      sAdsIkInkStorageTank[iL_Counter].sI_EnableMaintenance.bO_CommandCanEx  :=     sAdsIkInkStorageTank[iL_Counter].sI_EnableBalance.bI_Command
                                                                                AND NOT sAdsIkInkStorageTank[iL_Counter].sI_EnableMaintenance.bI_Command
                                                                                AND NOT sAdsIkInkStorageTank[iL_Counter].sI_EnableMaintenance.bO_CommandExec;
(*      bL_MessageWarning[iL_Counter] := (   sAdsIkInkStorageTank[iL_Counter].bO_StorageTankWarning
                                        OR (    sAdsIkInkStorageTank[iL_Counter].bO_StorageTankError
                                            AND NOT sAdsIkInkStorageTank[iL_Counter].bI_EnableStorageTank));*)
      bL_MessageWarning[iL_Counter] := (    sAdsIkInkStorageTank[iL_Counter].bO_StorageTankWarning
                                        AND sAdsIkInkStorageTank[iL_Counter].bI_EnableStorageTank);
      bL_MessageError  [iL_Counter] := (    sAdsIkInkStorageTank[iL_Counter].bO_StorageTankError
                                        AND sAdsIkInkStorageTank[iL_Counter].bI_EnableStorageTank);
    END_FOR; (*FOR iL_Counter := 1 TO iCIk_NB_INKBALANCE DO*)

    FOR iL_Counter := 1 TO iCIk_NB_INKSTORAGE_TANK DO
      (*Storage Messages*)
      fB_BalanceMsgHandler[iL_Counter]();	(*Call to check for blocked access*)

      fb_BalanceMsg[iL_Counter, 1](bI_Status := fb_BalanceLink.wO_ErrorCodeChannel[iL_Counter].1);
      fb_BalanceMsg[iL_Counter, 2](bI_Status := fb_BalanceLink.wO_ErrorCodeChannel[iL_Counter].2);
      fb_BalanceMsg[iL_Counter, 3](bI_Status := fb_BalanceLink.wO_ErrorCodeChannel[iL_Counter].3);
      fb_BalanceMsg[iL_Counter, 4](bI_Status := fb_BalanceLink.wO_ErrorCodeChannel[iL_Counter].4);
      fb_BalanceMsg[iL_Counter, 5](bI_Status := FALSE);
      fb_BalanceMsg[iL_Counter, 6](bI_Status := FALSE);
      fb_BalanceMsg[iL_Counter, 7](bI_Status := FALSE);
      fb_BalanceMsg[iL_Counter, 8](bI_Status := bL_MessageWarning[iL_Counter]);
      fb_BalanceMsg[iL_Counter, 9](bI_Status := bL_MessageError  [iL_Counter]);
      fb_BalanceMsg[iL_Counter,10](bI_Status := FALSE);
      fb_BalanceMsg[iL_Counter,11](bI_Status := FALSE);  (*InkStorageTankMixerNotWorking*)
      (*Storage tank level info message*)
      fb_BalanceMsg[iL_Counter,12](bI_Status :=     (   sAdsIkInkStorageTank[iL_Counter].bO_StorageTankWarning
                                                     OR sAdsIkInkStorageTank[iL_Counter].bO_StorageTankError)
                                                AND NOT sAdsIkInkStorageTank[iL_Counter].cO_StatusStorageTank.eO_Activ);
      fB_BalanceMsg[iL_Counter,13](bI_Status :=     fb_BarcodeStoragetank.bO_LabelScanNeeded[iL_Counter]
                                                AND sAdsIkInkStorageTank[iL_Counter].cO_StatusStorageTank.eO_Activ);
      fB_BalanceMsg[iL_Counter,14](bI_Status :=     fb_BarcodeStoragetank.bO_LabelScanFalse [iL_Counter]
                                                AND sAdsIkInkStorageTank[iL_Counter].cO_StatusStorageTank.eO_Activ);
      fB_BalanceMsg[iL_Counter,15](bI_Status :=     NOT fb_Storagetank[iL_Counter].bI_HtAssignedToStorage
                                                AND sAdsIkInkStorageTank[iL_Counter].cO_StatusStorageTank.eO_Activ);

      fb_MsgQueueStorage[iL_Counter]();

    END_FOR;
  END_IF; (*IF bCIk_BALANCE_EXISTING THEN*)

  (*Set fO_StorageTankLevelPercent of conservation tank with bO_TankCleanerLevelEmpty*)
  IF bO_TankCleanerLevelEmpty THEN
    sAdsIkInkStorageTank[iCIk_NB_INKSTORAGE_TANK].fO_StorageTankLevelPercent.fO_Val := 0;
  ELSE
    sAdsIkInkStorageTank[iCIk_NB_INKSTORAGE_TANK].fO_StorageTankLevelPercent.fO_Val := 100;
END_IF
  
END_IF; (*Else when init Ok*)


(*Global status*)
bO_InkSystemOk :=     bO_VacuumOk
                  AND bO_TemperatureOk
                //AND bO_StorageTankOk
                  AND (NOT bO_CommandPrintlineExec[1] OR NOT bL_Engaged[1])
                  AND (NOT bO_CommandPrintlineExec[2] OR NOT bL_Engaged[2]);

IF sL_SystemCmd.bSleep THEN
  bO_InkStorageTankOk := TRUE;
ELSE
  bO_InkStorageTankOk := FALSE;
  FOR iL_Counter := 1 TO iCIk_NB_INKSTORAGE_TANK DO
    IF bCIk_INKSTORAGE_TANK_EXIST[iL_Counter] THEN
      bO_InkStorageTankOk := bO_InkStorageTankOk OR sAdsIkInkStorageTank[iL_Counter].bI_EnableStorageTank;
    END_IF;
  END_FOR;
END_IF;

(*WcState: 0 = Data valid, 1 = Data invalid*)
bO_TotalWcState     :=     bI_Pressure1WcState
                        OR bI_Pressure2WcState
                        OR bI_SubPressureWcState[1]
                        OR bI_Temperature1WcState
                        OR bI_InkLevel1WcState;


(********************************* END OF PRG ****************************************************)

ACTION AutoFlushingDevice:
IF aI_FlushingSafePattern = 'SAFE' THEN
  bL_FlushingUnlock      := TRUE;
ELSE
  aI_FlushingSafePattern := 'LOCKED';
  bL_FlushingUnlock      := FALSE;
END_IF;
fb_FTrigFlushingActive(CLK:= bL_FlushingActive);
fb_TonFlushingUnlock(IN := bL_FlushingUnlock AND (iL_FlushingState = 0), PT := T#180S);
IF fb_TonFlushingUnlock.Q OR fb_FTrigFlushingActive.Q THEN
  aI_FlushingSafePattern := 'LOCKED';
  bL_FlushingHtEmpty     := FALSE;
END_IF

fb_FlushingReturnFlowTimer( bI_Reset    := (iL_FlushingState = 0)
                          , bI_In       :=    fb_ReturnFlow[iCIk_MAP_HEADERTANK_RETURN_FLOW[PRG_INK.iL_SelHeaderTankFlushing]].fb_ReturnFlowPump.bOKp_EnablePump
                                           OR bO_FlushingReturnPump[iCIk_MAP_HEADERTANK_RETURN_FLOW[PRG_INK.iL_SelHeaderTankFlushing]]
                          , lIO_Seconds := lL_OpCounterReturnFlowSeconds
                          , lIO_Cycles  := lL_OpCounterReturnFlowCycles);

(*Return if function is not unlocked.*)
IF NOT bL_FlushingUnlock THEN
  RETURN;
END_IF

CASE iL_FlushingState OF
0:  (*Idle*)
  aL_FlushingState := 'Idle';

  IF     bL_FlushingActivate 
     AND bL_FlushingHtEmpty 
     AND sAdsIkHeaderTank[PRG_INK.iL_SelHeaderTankFlushing].sI_ActivateCleaner.bO_CommandCanEx
     AND NOT sAdsIkHeaderTank[PRG_INK.iL_SelHeaderTankFlushing].bI_EnableFillInk
  THEN
    bL_FlushingActive := TRUE;

    iL_FlushingState  := 1;
  ELSE
    bL_FlushingStop     := FALSE;
    bL_FlushingActivate := FALSE;
    bL_FlushingActive   := FALSE;
    bL_FlushingActiveHt         [PRG_INK.iL_SelHeaderTankFlushing] := FALSE;
    bL_FlushingReturnFlowRequest[PRG_INK.iL_SelHeaderTankFlushing] := FALSE;
    sAdsIkHeaderTank[PRG_INK.iL_SelHeaderTankFlushing].sI_ActivateCleaner.bI_Command := FALSE;
	END_IF

1:  (*Start fill cleaner*)
  aL_FlushingState := 'Start fill cleaner';

  sAdsIkHeaderTank[PRG_INK.iL_SelHeaderTankFlushing].sI_ActivateCleaner.bI_Command := TRUE;
  
  IF sAdsIkHeaderTank[PRG_INK.iL_SelHeaderTankFlushing].sI_ActivateCleaner.bO_CommandExec THEN
    sAdsIkHeaderTank[PRG_INK.iL_SelHeaderTankFlushing].sI_ActivateCleaner.bI_Command := FALSE;
    bL_FlushingActiveHt[PRG_INK.iL_SelHeaderTankFlushing] := TRUE;

    iL_FlushingState := 2;
	END_IF
  
  IF bL_FlushingStop THEN
    sAdsIkHeaderTank[PRG_INK.iL_SelHeaderTankFlushing].sI_ActivateCleaner.bI_Command := FALSE;

    iL_FlushingState := 5;
	END_IF
  
2:  (*Fill cleaner*)
  aL_FlushingState := 'Fill cleaner';

  IF NOT sAdsIkHeaderTank[PRG_INK.iL_SelHeaderTankFlushing].sI_ActivateCleaner.bO_CommandExec THEN
    iL_FlushingState := 3;
	END_IF
  
  IF bL_FlushingStop THEN
    iL_FlushingState := 5;
	END_IF
  
3:  (*Start empty cleaner*)
  aL_FlushingState := 'Start empty cleaner';

  bL_FlushingReturnFlowRequest[PRG_INK.iL_SelHeaderTankFlushing] := TRUE;
  
  IF    fb_ReturnFlow[iCIk_MAP_HEADERTANK_RETURN_FLOW[PRG_INK.iL_SelHeaderTankFlushing]].fb_ReturnFlowPump.bOKp_EnablePump 
     OR bO_FlushingReturnPump[iCIk_MAP_HEADERTANK_RETURN_FLOW[PRG_INK.iL_SelHeaderTankFlushing]]
  THEN
    iL_FlushingState := 4;
	END_IF

  IF bL_FlushingStop THEN
    bL_FlushingReturnFlowRequest[PRG_INK.iL_SelHeaderTankFlushing] := FALSE;

    iL_FlushingState := 5;
	END_IF
  
4:  (*Empty cleaner*)
  aL_FlushingState := 'Empty cleaner';

  IF lL_OpCounterReturnFlowSeconds >= lL_TimeFlushingReturnFlow THEN
    bL_FlushingReturnFlowRequest[PRG_INK.iL_SelHeaderTankFlushing] := FALSE;
    bL_FlushingActiveHt         [PRG_INK.iL_SelHeaderTankFlushing] := FALSE;

    iL_FlushingState := 0;
	END_IF

  IF bL_FlushingStop THEN
    bL_FlushingReturnFlowRequest[PRG_INK.iL_SelHeaderTankFlushing] := FALSE;

    iL_FlushingState := 5;
	END_IF
  
5:  (*Abort*)
  aL_FlushingState := 'Abort';

  IF     NOT sAdsIkHeaderTank[PRG_INK.iL_SelHeaderTankFlushing].sI_ActivateCleaner.bO_CommandExec
     AND (   NOT fb_ReturnFlow[iCIk_MAP_HEADERTANK_RETURN_FLOW[PRG_INK.iL_SelHeaderTankFlushing]].fb_ReturnFlowPump.bOKp_EnablePump
          OR NOT bO_FlushingReturnPump[iCIk_MAP_HEADERTANK_RETURN_FLOW[PRG_INK.iL_SelHeaderTankFlushing]])
  THEN
    bL_FlushingStop     := FALSE;
    bL_FlushingActivate := FALSE;

    iL_FlushingState := 0;
	END_IF

END_CASE
END_ACTION

ACTION Init:
(*************************************************************************************************)
(* --- Module preprarations --- *)


(*GENERAL*)
(*************************************************************************************************)
(*System init*)
CASE cL_State OF

  cL_INIT : 		(*First init*)

                // Get system reference
                ISystemBase := PRG_SYSTEMBASE.getSystemBaseInterface();
                IF ISystemBase = 0 THEN RETURN; END_IF
                // Wait until system(base) is booted
                IF ISystemBase.bBooting THEN RETURN; END_IF
                
                // Command / Status interface
                PRG_SYSTEMBASE.getSystemCmdStatusInterface(iSystemCmd=>iSystemCmd, iSystemStatus=>iSystemStatus);
                
                // Build mapping information for ADS
                Mapping();
                
                // Register module to system
                pModuleDef := ISystemBase.regModule(
                  pAdsInfo:=ADR(sC_Ads_Info),
                  pMapInfo:=ADR(sMappingInfo)
                );
                IF pModuleDef = 0 THEN RETURN; END_IF

                Fb_RegToAry.iI_ActElem := 0;   (*init module's block mapping array*)
                Fb_RegToAry.sI_Parent := FC_CREATE_ARYPTR(ADR(sL_MOD_MAP), SIZEOF(sL_MOD_MAP)/SIZEOF(sL_MOD_MAP[1]), SIZEOF(sL_MOD_MAP[1]));

                iMachineInk[1] := PRG_MACHINE.fb_InterfaceMachineInk[1];
                iMachineInk[2] := PRG_MACHINE.fb_InterfaceMachineInk[2];

                cL_State := cL_INIT_PRG;

  cL_INIT_PRG :	(*Program call init*)

                FOR iL_CounterDgas := 1 TO iCIk_NB_DGAS DO
                  ;
                END_FOR;

                FOR iL_CounterMenc := 1 TO iCIk_NB_MENC DO
                  ;
                END_FOR

                FOR iL_CounterSubMenc := 1 TO iCIk_NB_SUB_MENC DO
                  ;
                END_FOR

                bL_RemVar_Init := TRUE;    (* Write variables by remanent variables *)
                RemVar();

                cL_State := cL_INIT_OK;

  cL_INIT_OK: 	(*First init ok*)
                bO_InitOk := TRUE;

END_CASE;



(*************************************************************************************************)
(*ADS Structures Init*)
(*************************************************************************************************)

(*INK TABLE*)
(*************************************************************************************************)
sL_InkTable[1].iI_ColorID := 0; sL_InkTable[1].aI_ColorName := sC_Config_I.aC_HEADERTANK_NAME_DETAIL[1]; sL_InkTable[1].lI_ColorRGB := 16#FFFFFF;
sL_InkTable[2].iI_ColorID := 0; sL_InkTable[2].aI_ColorName := sC_Config_I.aC_HEADERTANK_NAME_DETAIL[2]; sL_InkTable[2].lI_ColorRGB := 16#FFFFFF;
sL_InkTable[3].iI_ColorID := 1; sL_InkTable[3].aI_ColorName := sC_Config_I.aC_HEADERTANK_NAME_DETAIL[3]; sL_InkTable[3].lI_ColorRGB := 16#FFFFFF;
sL_InkTable[4].iI_ColorID := 1; sL_InkTable[4].aI_ColorName := sC_Config_I.aC_HEADERTANK_NAME_DETAIL[4]; sL_InkTable[4].lI_ColorRGB := 16#FFFFFF;


(*DEGASSING*)
(*************************************************************************************************)
(*Pneumatic Controller Board CB1*)
(*generate block ads name*)
FOR iL_Counter := 1 TO iCIk_NB_DGAS DO
  aL_Name := sC_Config_I.aC_DGAS_NAME;
  IF sC_Config_I.aC_DGAS_NAME_DETAIL[iL_Counter] <> '' THEN
    aL_Name := CONCAT(aL_Name, CONCAT(' - ', sC_Config_I.aC_DGAS_NAME_DETAIL[iL_Counter]));
  ELSE
    aL_Name := CONCAT(aL_Name, INT_TO_STRING(iL_Counter));
  END_IF
  sAdsIkDgas[iL_Counter].aO_Name := aL_Name;
END_FOR;

sAdsIkDgas[eIk_DGAS1].sI_PressSet.aC_Type := sC_Config_I.aC_DGAS1_PRESS_TYPE;
sAdsIkDgas[eIk_DGAS1].sI_PressSet.aC_Unit := sC_Config_I.aC_DGAS1_PRESS_UNIT;
sAdsIkDgas[eIk_DGAS1].sI_PressSet.fC_Min  := sC_Config_I.fL_DGAS1_PRESS_SET_MIN;
sAdsIkDgas[eIk_DGAS1].sI_PressSet.fC_Max  := sC_Config_I.fL_DGAS1_PRESS_SET_MAX;

sAdsIkDgas[eIk_DGAS1].sO_PressAct.aC_Type := sC_Config_I.aC_DGAS1_PRESS_TYPE;
sAdsIkDgas[eIk_DGAS1].sO_PressAct.aC_Unit := sC_Config_I.aC_DGAS1_PRESS_UNIT;
sAdsIkDgas[eIk_DGAS1].sO_PressAct.fC_Min  := sC_Config_I.fL_DGAS1_PRESS_ACT_MIN;
sAdsIkDgas[eIk_DGAS1].sO_PressAct.fC_Max  := sC_Config_I.fL_DGAS1_PRESS_ACT_MAX;

sAdsIkDgas[eIk_DGAS1].sI_AckPression.bO_CommandExist := TRUE;


(*MENISCUS*)
(*************************************************************************************************)
(*generate block ads name*)
FOR iL_Counter := 1 TO iCIk_NB_MENC DO
  aL_Name := sC_Config_I.aC_MENC_NAME;
  IF sC_Config_I.aC_MENC_NAME_DETAIL[iL_Counter] <> '' THEN
    aL_Name := CONCAT(aL_Name, CONCAT(' - ', sC_Config_I.aC_MENC_NAME_DETAIL[iL_Counter]));
  ELSE
    aL_Name := CONCAT(aL_Name, INT_TO_STRING(iL_Counter));
  END_IF
  sAdsIkMenc[iL_Counter].aO_Name := aL_Name;

  sAdsIkMenc[iL_Counter].sI_PressSet.aC_Type := sC_Config_I.aC_MENC_PRESS_TYPE;
  sAdsIkMenc[iL_Counter].sI_PressSet.aC_Unit := sC_Config_I.aC_MENC_PRESS_UNIT;
  sAdsIkMenc[iL_Counter].sI_PressSet.fC_Min  := sC_Config_I.fL_MENC_PRESS_SET_MIN;
  sAdsIkMenc[iL_Counter].sI_PressSet.fC_Max  := sC_Config_I.fL_MENC_PRESS_SET_MAX;

  sAdsIkMenc[iL_Counter].sO_PressAct.aC_Type := sC_Config_I.aC_MENC_PRESS_TYPE;
  sAdsIkMenc[iL_Counter].sO_PressAct.aC_Unit := sC_Config_I.aC_MENC_PRESS_UNIT;
  sAdsIkMenc[iL_Counter].sO_PressAct.fC_Min  := sC_Config_I.fL_MENC_PRESS_ACT_MIN;
  sAdsIkMenc[iL_Counter].sO_PressAct.fC_Max  := sC_Config_I.fL_MENC_PRESS_ACT_MAX;

  sAdsIkMenc[iL_Counter].sI_AckPression.bO_CommandExist := TRUE;
END_FOR;


(*SUB MENISCUS*)
(*************************************************************************************************)
(*Sub meniscus starts behind the meniscus*)
(*generate block ads name*)
FOR iL_CounterSubMenc := 1 TO iCIk_NB_SUB_MENC DO
  aL_Name := sC_Config_I.aC_SUB_MENC_NAME;
  IF sC_Config_I.aC_SUB_MENC_NAME_DETAIL[iL_CounterSubMenc] <> '' THEN
    aL_Name := CONCAT(aL_Name, CONCAT(' - ', sC_Config_I.aC_SUB_MENC_NAME_DETAIL[iL_CounterSubMenc]));
  ELSE
    aL_Name := CONCAT(aL_Name, INT_TO_STRING(iCIk_NB_MENC + iL_CounterSubMenc));
  END_IF
  sAdsIkMenc[iCIk_NB_MENC + iL_CounterSubMenc].aO_Name := aL_Name;

  sAdsIkMenc[iCIk_NB_MENC + iL_CounterSubMenc].sI_PressSet.aC_Type := sC_Config_I.aC_SUB_MENC_PRESS_TYPE;
  sAdsIkMenc[iCIk_NB_MENC + iL_CounterSubMenc].sI_PressSet.aC_Unit := sC_Config_I.aC_SUB_MENC_PRESS_UNIT;
  sAdsIkMenc[iCIk_NB_MENC + iL_CounterSubMenc].sI_PressSet.fC_Min  := sC_Config_I.fL_SUB_MENC_PRESS_SET_MIN;
  sAdsIkMenc[iCIk_NB_MENC + iL_CounterSubMenc].sI_PressSet.fC_Max  := sC_Config_I.fL_SUB_MENC_PRESS_SET_MAX;

  sAdsIkMenc[iCIk_NB_MENC + iL_CounterSubMenc].sO_PressAct.aC_Type := sC_Config_I.aC_SUB_MENC_PRESS_TYPE;
  sAdsIkMenc[iCIk_NB_MENC + iL_CounterSubMenc].sO_PressAct.aC_Unit := sC_Config_I.aC_SUB_MENC_PRESS_UNIT;
  sAdsIkMenc[iCIk_NB_MENC + iL_CounterSubMenc].sO_PressAct.fC_Min  := sC_Config_I.fL_SUB_MENC_PRESS_ACT_MIN;
  sAdsIkMenc[iCIk_NB_MENC + iL_CounterSubMenc].sO_PressAct.fC_Max  := sC_Config_I.fL_SUB_MENC_PRESS_ACT_MAX;

  sAdsIkMenc[iCIk_NB_MENC + iL_CounterSubMenc].sI_AckPression.bO_CommandExist := TRUE;

  //sAdsIkMenc[iCIk_NB_MENC + iL_CounterSubMenc].iO_ColorId          := x;
END_FOR;


(*PURGE*)
(*************************************************************************************************)
(*generate block ads name*)
FOR iL_Counter := 1 TO iCIk_NB_PURGE_CONTR DO
  aL_Name := sC_Config_I.aC_PURGE_NAME;
  IF sC_Config_I.aC_PURGE_NAME_DETAIL[iL_Counter] <> '' THEN
    aL_Name := CONCAT(aL_Name, CONCAT(' - ', sC_Config_I.aC_PURGE_NAME_DETAIL[iL_Counter]));
  ELSE
    aL_Name := CONCAT(aL_Name, INT_TO_STRING(iL_Counter));
  END_IF
  sAdsIkPurgeController[iL_Counter].aO_Name := aL_Name;

  sAdsIkPurgeController[iL_Counter].sI_ActivatePurge.bO_CommandCanEx := TRUE;
  sAdsIkPurgeController[iL_Counter].sI_ActivatePurge.bO_CommandExist := TRUE;
END_FOR;

FOR iL_Counter := 1 TO iCIk_NB_PURGE_GROUP DO
  (*generate block ads name*)
  aL_Name := sC_Config_I.aC_PURGE_GROUP_NAME;
  IF sC_Config_I.aC_PURGE_GROUP_NAME_DETAIL[iL_Counter] <> '' THEN
    aL_Name := CONCAT(aL_Name, CONCAT(' - ', sC_Config_I.aC_PURGE_GROUP_NAME_DETAIL[iL_Counter]));
  ELSE
    aL_Name := CONCAT(aL_Name, INT_TO_STRING(iL_Counter));
  END_IF
  sAdsIkPurgeGroup[iL_Counter].aO_Name := aL_Name;

  sAdsIkPurgeGroup[iL_Counter].cO_Status.eO_Avbl      := TRUE;
  sAdsIkPurgeGroup[iL_Counter].cO_ValveStatus.eO_Avbl := TRUE;
END_FOR


(*INK*)
(*************************************************************************************************)
FOR iL_Counter := 1 TO iCIk_NB_INK_PUMPS DO
  (*generate block ads name*)
  aL_Name := sC_Config_I.aC_INKPUMP_NAME;
  IF sC_Config_I.aC_INKPUMP_NAME_DETAIL[iL_Counter] <> '' THEN
    aL_Name := CONCAT(aL_Name, CONCAT(' - ', sC_Config_I.aC_INKPUMP_NAME_DETAIL[iL_Counter]));
  ELSE
    aL_Name := CONCAT(aL_Name, INT_TO_STRING(iL_Counter));
  END_IF
  sAdsIkInkPump[iL_Counter].aO_Name := aL_Name;

  sAdsIkInkPump[iL_Counter].sI_InkPumpSpeedSet.aC_Type := sC_Config_I.aC_INKPUMP_SPEED_TYPE;
  sAdsIkInkPump[iL_Counter].sI_InkPumpSpeedSet.aC_Unit := sC_Config_I.aC_INKPUMP_SPEED_UNIT;
  sAdsIkInkPump[iL_Counter].sI_InkPumpSpeedSet.lC_Min  := sC_Config_I.lL_INKPUMP_SPEED_SET_MIN;
  sAdsIkInkPump[iL_Counter].sI_InkPumpSpeedSet.lC_Max  := sC_Config_I.lL_INKPUMP_SPEED_SET_MAX;
END_FOR

FOR iL_Counter := 1 TO iCIk_NB_HEADERTANK DO
  (*IF bCIk_HEADERTANK_EXIST[iL_Counter] THEN*)
    (*generate block ads name*)
    aL_Name := sC_Config_I.aC_HEADERTANK_NAME;
    IF sC_Config_I.aC_HEADERTANK_NAME_DETAIL[iL_Counter] <> '' THEN
      aL_Name := CONCAT(aL_Name, CONCAT(' - ', sC_Config_I.aC_HEADERTANK_NAME_DETAIL[iL_Counter]));
    ELSE
      aL_Name := CONCAT(aL_Name, INT_TO_STRING(iL_Counter));
    END_IF
    sAdsIkHeaderTank[iL_Counter].aO_Name := aL_Name;

		sAdsIkHeaderTank[iL_Counter].sI_StoragetankAssignment.bC_Exist    := TRUE;
		sAdsIkHeaderTank[iL_Counter].sO_ActStoragetankAssignment.bC_Exist := TRUE;

		(*un-/fill ink*)
		sAdsIkHeaderTank[iL_Counter].bO_EnableFillInkCanEn               := bCIk_HEADERTANK_EXIST[iL_Counter];
		sAdsIkHeaderTank[iL_Counter].bO_EnableUnFillInkCanEn             := bCIk_HEADERTANK_EXIST[iL_Counter];
		sAdsIkHeaderTank[iL_Counter].cO_StatusFillInk.eO_Avbl            := bCIk_HEADERTANK_EXIST[iL_Counter];
		sAdsIkHeaderTank[iL_Counter].cO_StatusUnFillInk.eO_Avbl          := bCIk_HEADERTANK_EXIST[iL_Counter];

		sAdsIkHeaderTank[iL_Counter].sI_ActivateCleaner.bO_CommandCanEx  := bCIk_HEADERTANK_FILL_CLEANER[iL_Counter];
		sAdsIkHeaderTank[iL_Counter].sI_ActivateRefuse.bO_CommandCanEx   := bCIk_HEADERTANK_REFUSE      [iL_Counter];
		sAdsIkHeaderTank[iL_Counter].sI_ActivateExchange.bO_CommandCanEx := FALSE;

		sAdsIkHeaderTank[iL_Counter].sI_ActivateCleaner.bO_CommandExist	 := bCIk_HEADERTANK_FILL_CLEANER[iL_Counter];
		sAdsIkHeaderTank[iL_Counter].sI_ActivateRefuse.bO_CommandExist	 := bCIk_HEADERTANK_REFUSE      [iL_Counter];
		sAdsIkHeaderTank[iL_Counter].sI_ActivateExchange.bO_CommandExist := FALSE;

    sAdsIkHeaderTank[iL_Counter].sI_CommandChange.bO_CommandExist    := bCIk_HEADERTANK_CHANGE      [iL_Counter];

		(*error ack exist*)
		sAdsIkHeaderTank[iL_Counter].sI_AckFillInk.bO_CommandExist       := TRUE;

		(*tank heater*)
		sAdsIkHeaderTank[iL_Counter].sI_TankHeaterSet.bC_Exist   := FALSE;
		sAdsIkHeaderTank[iL_Counter].sI_TankHeaterSet.aC_Type    := sC_Config_I.aC_TEMP_TYPE;
		sAdsIkHeaderTank[iL_Counter].sI_TankHeaterSet.aC_Unit    := sC_Config_I.aC_TEMP_UNIT;
		sAdsIkHeaderTank[iL_Counter].sI_TankHeaterSet.fC_Min     := sC_Config_I.fL_TEMP_SET_VAL_MIN;
		sAdsIkHeaderTank[iL_Counter].sI_TankHeaterSet.fC_Max     := sC_Config_I.fL_TEMP_SET_VAL_MAX;

		sAdsIkHeaderTank[iL_Counter].sO_TankHeaterAct.bC_Exist   := FALSE;
		sAdsIkHeaderTank[iL_Counter].sO_TankHeaterAct.aC_Type    := sC_Config_I.aC_TEMP_TYPE;
		sAdsIkHeaderTank[iL_Counter].sO_TankHeaterAct.aC_Unit    := sC_Config_I.aC_TEMP_UNIT;
    sAdsIkHeaderTank[iL_Counter].sO_TankHeaterAct.fC_Min     := sC_Config_I.fL_TEMP_ACT_VAL_MIN;
    sAdsIkHeaderTank[iL_Counter].sO_TankHeaterAct.fC_Max     := sC_Config_I.fL_TEMP_ACT_VAL_MAX;

		sAdsIkHeaderTank[iL_Counter].bO_EnableTankHeaterCanEn    := FALSE;
		sAdsIkHeaderTank[iL_Counter].cO_StatusTankHeater.eO_Avbl := FALSE;
	(*END_IF*)
END_FOR

FOR iL_Counter := 1 TO iCIk_NB_HEADERTANK_GROUP DO
  (*generate block ads name*)
  aL_Name := sC_Config_I.aC_HEADERTANKGROUP_NAME;
  IF sC_Config_I.aC_HEADERTANKGROUP_NAME_DETAIL[iL_Counter] <> '' THEN
    aL_Name := CONCAT(aL_Name, CONCAT(' - ', sC_Config_I.aC_HEADERTANKGROUP_NAME_DETAIL[iL_Counter]));
  ELSE
    aL_Name := CONCAT(aL_Name, INT_TO_STRING(iL_Counter));
  END_IF
  sAdsIkHeaderTankGroup[iL_Counter].aO_Name := aL_Name;

  sAdsIkHeaderTankGroup[iL_Counter].sI_CommandChangeInk.bO_CommandExist := TRUE;
  sAdsIkHeaderTankGroup[iL_Counter].sI_CommandChangeInk.bO_CommandCanEx := TRUE;
  sAdsIkHeaderTankGroup[iL_Counter].sI_CommandEmptyInk.bO_CommandExist  := FALSE;
  sAdsIkHeaderTankGroup[iL_Counter].sI_CommandEmptyInk.bO_CommandCanEx  := FALSE;
END_FOR


(*TEMP*)
(*************************************************************************************************)
FOR iL_Counter := 1 TO iCIk_NB_TEMP_CONTR DO
  (*generate block ads name*)
  aL_Name := sC_Config_I.aC_TEMP_NAME;
  IF sC_Config_I.aC_TEMP_NAME_DETAIL[iL_Counter] <> '' THEN
    aL_Name := CONCAT(aL_Name, CONCAT(' - ', sC_Config_I.aC_TEMP_NAME_DETAIL[iL_Counter]));
  ELSE
    aL_Name := CONCAT(aL_Name, INT_TO_STRING(iL_Counter));
  END_IF
  sAdsIkHeater[iL_Counter].aO_Name := aL_Name;

  sAdsIkHeater[iL_Counter].sI_HeaterSet.aC_Type    := sC_Config_I.aC_TEMP_TYPE;
  sAdsIkHeater[iL_Counter].sI_HeaterSet.aC_Unit    := sC_Config_I.aC_TEMP_UNIT;
  sAdsIkHeater[iL_Counter].sI_HeaterSet.fC_Min     := sC_Config_I.fL_TEMP_SET_VAL_MIN;
  sAdsIkHeater[iL_Counter].sI_HeaterSet.fC_Max     := sC_Config_I.fL_TEMP_SET_VAL_MAX;

  sAdsIkHeater[iL_Counter].sO_HeaterAct.aC_Type    := sC_Config_I.aC_TEMP_TYPE;
  sAdsIkHeater[iL_Counter].sO_HeaterAct.aC_Unit    := sC_Config_I.aC_TEMP_UNIT;
  sAdsIkHeater[iL_Counter].sO_HeaterAct.fC_Min     := sC_Config_I.fL_TEMP_ACT_VAL_MIN;
  sAdsIkHeater[iL_Counter].sO_HeaterAct.fC_Max     := sC_Config_I.fL_TEMP_ACT_VAL_MAX;

  sAdsIkHeater[iL_Counter].bO_EnableHeaterCanEn    := TRUE;
  sAdsIkHeater[iL_Counter].cO_StatusHeater.eO_Avbl := TRUE;
END_FOR


(* STORAGE TANK *)
(**********************************************************************************)
FOR iL_Counter := 1 TO iCIk_NB_INKSTORAGE_TANK DO
  (*generate block ads name*)
  aL_Name := sC_Config_I.aC_STORAGETANK_NAME;
  IF sC_Config_I.aC_STORAGETANK_NAME_DETAIL[iL_Counter] <> '' THEN
    aL_Name := CONCAT(aL_Name, CONCAT(' - ', sC_Config_I.aC_STORAGETANK_NAME_DETAIL[iL_Counter]));
  ELSE
    aL_Name := CONCAT(aL_Name, INT_TO_STRING(iL_Counter));
  END_IF
  sAdsIkInkStorageTank[iL_Counter].aO_Name := aL_Name;

  (*Special storage tank for conservation*)
  IF sC_Config_I.aC_STORAGETANK_NAME_DETAIL[iL_Counter] = sC_Config_I.aC_STORAGETANK_CONSERVATION THEN
    sAdsIkInkStorageTank[iL_Counter].bO_EnableStorageTankCanEn             := FALSE;
    sAdsIkInkStorageTank[iL_Counter].cO_StatusStorageTank.eO_Avbl          := FALSE;
    sAdsIkInkStorageTank[iL_Counter].sI_EnableMaintenance.bO_CommandCanEx  := FALSE;
    sAdsIkInkStorageTank[iL_Counter].sI_EnableMaintenance.bO_CommandExist  := FALSE;
    sAdsIkInkStorageTank[iL_Counter].fO_StorageTankLevelLiter.bC_Exist     := FALSE;
    sAdsIkInkStorageTank[iL_Counter].sI_MaintenanceTimeout.bC_Exist        := FALSE;
    
    (*Varnish parameter*)
    sAdsIkInkStorageTank[iL_Counter].bO_InkParameterExist                  := FALSE;
    sAdsIkInkStorageTank[iL_Counter].sI_InkParameter.sTemperature.aC_Type  := sC_Config_I.aC_TEMP_TYPE;
    sAdsIkInkStorageTank[iL_Counter].sI_InkParameter.sTemperature.aC_Unit  := sC_Config_I.aC_TEMP_UNIT;
    sAdsIkInkStorageTank[iL_Counter].sI_InkParameter.sTemperature.fC_Min   := sC_Config_I.fL_TEMP_SET_VAL_MIN;
    sAdsIkInkStorageTank[iL_Counter].sI_InkParameter.sTemperature.fC_Max   := sC_Config_I.fL_TEMP_SET_VAL_MAX;
    sAdsIkInkStorageTank[iL_Counter].sI_InkParameter.sMeniscus.aC_Type     := sC_Config_I.aC_SUB_MENC_PRESS_TYPE;
    sAdsIkInkStorageTank[iL_Counter].sI_InkParameter.sMeniscus.aC_Unit     := sC_Config_I.aC_SUB_MENC_PRESS_UNIT;
    sAdsIkInkStorageTank[iL_Counter].sI_InkParameter.sMeniscus.fC_Min      := sC_Config_I.fL_SUB_MENC_PRESS_SET_MIN;
    sAdsIkInkStorageTank[iL_Counter].sI_InkParameter.sMeniscus.fC_Max      := sC_Config_I.fL_SUB_MENC_PRESS_SET_MAX;
    sAdsIkInkStorageTank[iL_Counter].sI_InkParameter.sDensity.aC_Unit      := sC_Config_I.aC_STORAGETANK_DENSITY;
    sAdsIkInkStorageTank[iL_Counter].sI_InkParameter.sViscosity.aC_Unit    := sC_Config_I.aC_STORAGETANK_VISCOSITY;

    sAdsIkInkStorageTank[iL_Counter].sI_EnableBalance.bO_CommandCanEx      := FALSE;
    sAdsIkInkStorageTank[iL_Counter].sI_EnableBalance.bO_CommandExist      := FALSE;
    sAdsIkInkStorageTank[iL_Counter].cO_StatusBalance.eO_Avbl              := FALSE;
    sAdsIkInkStorageTank[iL_Counter].bO_SetZeroCanEx                       := FALSE;
  ELSE
    sAdsIkInkStorageTank[iL_Counter].bI_EnableStorageTank                  := TRUE;
    sAdsIkInkStorageTank[iL_Counter].bO_EnableStorageTankCanEn             := TRUE;
    sAdsIkInkStorageTank[iL_Counter].cO_StatusStorageTank.eO_Avbl          := FALSE;
  
    sAdsIkInkStorageTank[iL_Counter].sI_EnableMaintenance.bO_CommandCanEx  := TRUE;
    sAdsIkInkStorageTank[iL_Counter].sI_EnableMaintenance.bO_CommandExist  := TRUE;
  
    sAdsIkInkStorageTank[iL_Counter].fO_StorageTankLevelLiter.aC_Type      := sC_Config_I.aC_STORAGETANK_TYPE;
    sAdsIkInkStorageTank[iL_Counter].fO_StorageTankLevelLiter.aC_Unit      := sC_Config_I.aC_STORAGETANK_UNITLITER;
    sAdsIkInkStorageTank[iL_Counter].fO_StorageTankLevelPercent.aC_Type    := sC_Config_I.aC_STORAGETANK_TYPE;
    sAdsIkInkStorageTank[iL_Counter].fO_StorageTankLevelPercent.aC_Unit    := sC_Config_I.aC_STORAGETANK_UNITPERCENT;
  
    sAdsIkInkStorageTank[iL_Counter].sI_MaintenanceTimeout.aC_Type         := sC_Config_I.aC_STORAGETANK_MAINTENANCE_TYPE;
    sAdsIkInkStorageTank[iL_Counter].sI_MaintenanceTimeout.aC_Unit         := sC_Config_I.aC_STORAGETANK_MAINTENANCE_UNIT;
    sAdsIkInkStorageTank[iL_Counter].sI_MaintenanceTimeout.lC_Min          := sC_Config_I.lL_STORAGETANK_MAINTENANCE_SET_MIN;
    sAdsIkInkStorageTank[iL_Counter].sI_MaintenanceTimeout.lC_Max          := sC_Config_I.lL_STORAGETANK_MAINTENANCE_SET_MAX;
  
    (*Varnish parameter*)
    sAdsIkInkStorageTank[iL_Counter].bO_InkParameterExist                  := TRUE;
    sAdsIkInkStorageTank[iL_Counter].sI_InkParameter.sTemperature.aC_Type  := sC_Config_I.aC_TEMP_TYPE;
    sAdsIkInkStorageTank[iL_Counter].sI_InkParameter.sTemperature.aC_Unit  := sC_Config_I.aC_TEMP_UNIT;
    sAdsIkInkStorageTank[iL_Counter].sI_InkParameter.sTemperature.fC_Min   := sC_Config_I.fL_TEMP_SET_VAL_MIN;
    sAdsIkInkStorageTank[iL_Counter].sI_InkParameter.sTemperature.fC_Max   := sC_Config_I.fL_TEMP_SET_VAL_MAX;
    sAdsIkInkStorageTank[iL_Counter].sI_InkParameter.sMeniscus.aC_Type     := sC_Config_I.aC_SUB_MENC_PRESS_TYPE;
    sAdsIkInkStorageTank[iL_Counter].sI_InkParameter.sMeniscus.aC_Unit     := sC_Config_I.aC_SUB_MENC_PRESS_UNIT;
    sAdsIkInkStorageTank[iL_Counter].sI_InkParameter.sMeniscus.fC_Min      := sC_Config_I.fL_SUB_MENC_PRESS_SET_MIN;
    sAdsIkInkStorageTank[iL_Counter].sI_InkParameter.sMeniscus.fC_Max      := sC_Config_I.fL_SUB_MENC_PRESS_SET_MAX;
    sAdsIkInkStorageTank[iL_Counter].sI_InkParameter.sDensity.aC_Unit      := sC_Config_I.aC_STORAGETANK_DENSITY;
    sAdsIkInkStorageTank[iL_Counter].sI_InkParameter.sViscosity.aC_Unit    := sC_Config_I.aC_STORAGETANK_VISCOSITY;
  END_IF
END_FOR;

FOR iL_Counter := 1 TO iCIk_NB_INKSTORAGE_TANK DO
  (*Varnish parameter*)
  IF sAdsIkInkStorageTank[iL_Counter].bO_InkParameterExist THEN
    sAdsIkInkStorageTank[iL_Counter].sI_InkParameter.iScannerId          := sR_RemVar_I.lR_VarParamScannerId[iL_Counter];
    sAdsIkInkStorageTank[iL_Counter].sI_InkParameter.iIndex              := sR_RemVar_I.iR_VarParamIndex    [iL_Counter];
    sAdsIkInkStorageTank[iL_Counter].sI_InkParameter.sTemperature.fI_Val := sR_RemVar_I.fR_VarParamTemp     [iL_Counter];
    sAdsIkInkStorageTank[iL_Counter].sI_InkParameter.sMeniscus.fI_Val    := sR_RemVar_I.fR_VarParamMenc     [iL_Counter];
    sAdsIkInkStorageTank[iL_Counter].sI_InkParameter.aWaveform           := sR_RemVar_I.aR_VarParamWaveform [iL_Counter];
    sAdsIkInkStorageTank[iL_Counter].sI_InkParameter.iTimer              := sR_RemVar_I.iR_VarParamTimer    [iL_Counter];
    sAdsIkInkStorageTank[iL_Counter].sI_InkParameter.sDensity.fI_Val     := sR_RemVar_I.fR_VarParamDensity  [iL_Counter];
    sAdsIkInkStorageTank[iL_Counter].sI_InkParameter.sViscosity.fI_Val   := sR_RemVar_I.fR_VarParamViscosity[iL_Counter];
    sAdsIkInkStorageTank[iL_Counter].sI_InkParameter.iColorId            := sR_RemVar_I.iR_VarParamColorId  [iL_Counter];
    FOR iL_Counter2 := 1 TO 10 DO
      sAdsIkInkStorageTank[iL_Counter].sI_InkParameter.bCompatibility[iL_Counter2] := sR_RemVar_I.bR_VarParamCompatibility[iL_Counter, iL_Counter2];
    END_FOR;
  END_IF
END_FOR;


(* BALANCE *)
(*************************************************************************************************)
(* -------------- init of the channels -------------------- *)
FOR iL_Counter := 1 TO iCIk_NB_INKBALANCE DO
  sAdsIkInkStorageTank[iL_Counter].sI_EnableBalance.bI_Command      := TRUE;
	sAdsIkInkStorageTank[iL_Counter].sI_EnableBalance.bO_CommandCanEx := TRUE;
	sAdsIkInkStorageTank[iL_Counter].sI_EnableBalance.bO_CommandExist := TRUE;
	sAdsIkInkStorageTank[iL_Counter].cO_StatusBalance.eO_Avbl         := TRUE;
	sAdsIkInkStorageTank[iL_Counter].bO_SetZeroCanEx                  := TRUE;

	sAdsIkInkStorageTank[iL_Counter].sI_InkDensitySet.aC_Type         := sC_Config_I.aC_BALANCE_INKDENSITY_TYPE;
	sAdsIkInkStorageTank[iL_Counter].sI_InkDensitySet.aC_Unit         := sC_Config_I.aC_BALANCE_INKDENSITY_UNIT;
	sAdsIkInkStorageTank[iL_Counter].sI_InkDensitySet.fC_Min          := sC_Config_I.aC_BALANCE_INKDENSITY_SET_MIN;
	sAdsIkInkStorageTank[iL_Counter].sI_InkDensitySet.fC_Max          := sC_Config_I.aC_BALANCE_INKDENSITY_SET_MAX;

	sAdsIkInkStorageTank[iL_Counter].sI_CorrectionValue.aC_Type       := sC_Config_I.aC_BALANCE_CORRECTION_TYPE;
	sAdsIkInkStorageTank[iL_Counter].sI_CorrectionValue.aC_Unit       := sC_Config_I.aC_BALANCE_CORRECTION_UNIT;
	sAdsIkInkStorageTank[iL_Counter].sI_CorrectionValue.fC_Min        := sC_Config_I.aC_BALANCE_CORRECTION_SET_MIN;
	sAdsIkInkStorageTank[iL_Counter].sI_CorrectionValue.fC_Max        := sC_Config_I.aC_BALANCE_CORRECTION_SET_MAX;

	sAdsIkInkStorageTank[iL_Counter].sI_WarningLevelSet.aC_Type       := sC_Config_I.aC_BALANCE_WARNINGLEVEL_TYPE;
	sAdsIkInkStorageTank[iL_Counter].sI_WarningLevelSet.aC_Unit       := sC_Config_I.aC_BALANCE_WARNINGLEVEL_UNIT;
	sAdsIkInkStorageTank[iL_Counter].sI_WarningLevelSet.fC_Min        := sC_Config_I.aC_BALANCE_WARNINGLEVEL_SET_MIN;
	sAdsIkInkStorageTank[iL_Counter].sI_WarningLevelSet.fC_Max        := sC_Config_I.aC_BALANCE_WARNINGLEVEL_SET_MAX;

	sAdsIkInkStorageTank[iL_Counter].sI_ErrorlevelSet.aC_Type         := sC_Config_I.aC_BALANCE_ERRORLEVEL_TYPE;
	sAdsIkInkStorageTank[iL_Counter].sI_ErrorlevelSet.aC_Unit         := sC_Config_I.aC_BALANCE_ERRORLEVEL_UNIT;
	sAdsIkInkStorageTank[iL_Counter].sI_ErrorlevelSet.fC_Min          := sC_Config_I.aC_BALANCE_ERRORLEVEL_SET_MIN;
	sAdsIkInkStorageTank[iL_Counter].sI_ErrorlevelSet.fC_Max          := sC_Config_I.aC_BALANCE_ERRORLEVEL_SET_MAX;
END_FOR;


(*************************************************************************************************)
(*Function Blocks Init*)
(*************************************************************************************************)


(*neue Lib: new code*)
(*DEGASSING*)
(*************************************************************************************************)
FOR iL_CounterDgas := 1 TO iCIk_NB_DGAS DO
  iSystemCmd.registerForSleepUpdate(iObserver:=fb_DgasMencContr[iL_CounterDgas]);
  
  fb_DgasMencContr[iL_CounterDgas].iRequestMencMinus       := fb_DgasPumpMinus[iL_CounterDgas];
  fb_DgasMencContr[iL_CounterDgas].iRequestMencPlus        := fb_DgasValvePlus[iL_CounterDgas];
  fb_DgasMencContr[iL_CounterDgas].iPurgeController        := fb_PurgeControllerDummy;  (*PurgeBusy not relevant*)
  fb_DgasMencContr[iL_CounterDgas].pConf                   := sC_Config_I.cC_CONF_DGAS_CONTR;
  fb_DgasMencContr[iL_CounterDgas].mInit( pAdsIf         := ADR(sAdsIkDgas [iL_CounterDgas])        (*> ads reference*)
                                        , pMap           := ADR(sL_BLK_DGAS[iL_CounterDgas]));        (*> mapping definition reference*)
  fb_DgasPumpMinus[iL_CounterDgas].mInit( aI_Name        := 'Dgas pump');

  (*MainValve K111*)
  iSystemCmd.registerForSleepUpdate(iObserver:=fb_DgasMainValve[iL_CounterDgas]);
  fb_DgasMainValve[iL_CounterDgas].mEnable();
END_FOR;

(*MENISCUS*)
(*************************************************************************************************)
FOR iL_CounterMenc := 1 TO iCIk_NB_MENC DO
  iSystemCmd.registerForSleepUpdate(iObserver:=fb_MeniscusMencContr[iL_CounterMenc]);
  
  fb_MeniscusMencContr[iL_CounterMenc].iRequestMencMinus       := fb_MeniscusValveMinus[iL_CounterMenc];
  fb_MeniscusMencContr[iL_CounterMenc].iRequestMencPlus        := fb_MeniscusValvePlus [iL_CounterMenc];
  fb_MeniscusMencContr[iL_CounterMenc].iPurgeController        := fb_PurgeControllerDummy;  (*PurgeBusy not relevant*)
  fb_MeniscusMencContr[iL_CounterMenc].pConf                   := sC_Config_I.cC_CONF_MENC_CONTR;
  fb_MeniscusMencContr[iL_CounterMenc].mInit( pAdsIf         := ADR(sAdsIkMenc [iL_CounterMenc])        (*> ads reference*)
                                            , pMap           := ADR(sL_BLK_MENC[iL_CounterMenc]));      (*> mapping definition reference*)
END_FOR;
fb_MeniscusPump.mInit(aI_Name := 'Main meniscus pump');

(*SUB MENISCUS*)
(*************************************************************************************************)
FOR iL_CounterSubMenc := 1 TO iCIk_NB_SUB_MENC DO
  iSystemCmd.registerForSleepUpdate(iObserver:=fb_MeniscusMencContr[iCIk_NB_MENC + iL_CounterSubMenc]);
  
  fb_MeniscusMencContr[iCIk_NB_MENC + iL_CounterSubMenc].iRequestMencMinus       := fb_MeniscusValveMinus[iCIk_NB_MENC + iL_CounterSubMenc];
  fb_MeniscusMencContr[iCIk_NB_MENC + iL_CounterSubMenc].iRequestMencPlus        := fb_MeniscusValvePlus [iCIk_NB_MENC + iL_CounterSubMenc];
  fb_MeniscusMencContr[iCIk_NB_MENC + iL_CounterSubMenc].iPurgeController        := fb_PurgeControllerDummy;  (*PurgeBusy not relevant*)
  fb_MeniscusMencContr[iCIk_NB_MENC + iL_CounterSubMenc].pConf                   := sC_Config_I.cC_CONF_SUB_MENC_CONTR;
  fb_MeniscusMencContr[iCIk_NB_MENC + iL_CounterSubMenc].mInit( pAdsIf         := ADR(sAdsIkMenc [iCIk_NB_MENC + iL_CounterSubMenc])  (*> ads reference*)
                                                              , pMap           := ADR(sL_BLK_MENC[iCIk_NB_MENC + iL_CounterSubMenc]));  (*> mapping definition reference*)
END_FOR;


(*TEMP*)
(*************************************************************************************************)
(*Headertank heater*)
FOR iL_Counter := 1 TO iCIk_NB_TEMP_HYS DO
  iSystemCmd.registerForSleepUpdate(iObserver:=fb_TempControllerHys[iL_Counter]);
  iSystemCmd.registerForEmergencyUpdate(iObserver:=fb_TempControllerHys[iL_Counter]);

  fb_TempControllerHys[iL_Counter].mInit( pAdsIf         := ADR(sAdsIkHeater[iL_Counter]));           (*> ads reference*)
  fb_TempControllerHys[iL_Counter].mEnable();
END_FOR;


(*PURGE*)
(*************************************************************************************************)
FOR iL_Counter := 1 TO iCIk_NB_PURGE_CONTR DO
  fb_PurgeController[iL_Counter].iMachineInk       := PRG_MACHINE.iMachineInk[iL_Counter];
  fb_PurgeController[iL_Counter].iSubMencNeg       := fb_MeniscusMencContr[bCIk_MAP_PURGE_CONTR_SEQ_MENC_NEG[iL_Counter]];
  fb_PurgeController[iL_Counter].iSubMencPos       := fb_MeniscusMencContr[bCIk_MAP_PURGE_CONTR_SEQ_MENC_POS[iL_Counter]];
  fb_PurgeController[iL_Counter].pActivateSequence := bCIk_PURGE_CONTR_SEQUENCE[iL_Counter];
  fb_PurgeController[iL_Counter].pAirOk            := TRUE;
  fb_PurgeController[iL_Counter].mInit( pAdsIf         := ADR(sAdsIkPurgeController[iL_Counter])  (*> ads reference*)
                                      , pMap           := ADR(sL_BLK_PURGE_CONTR   [iL_Counter]));  (*> mapping definition reference*)
END_FOR

FOR iL_Counter := 1 TO iCIk_NB_PURGE_GROUP DO
  fb_PurgeGroup     [iL_Counter].mInit( pAdsIf         := ADR(sAdsIkPurgeGroup  [iL_Counter])     (*> ads reference*)
                                      , pMap           := ADR(sL_BLK_PURGE_GROUP[iL_Counter]));     (*> mapping definition reference*)

  IF cL_State = cL_INIT_PRG THEN
    fb_PurgeController[cCIk_MAP_PURGE_GROUP_CONTR[iL_Counter]].mRegisterGroup(fb_PurgeGroup[iL_Counter]);
  END_IF
END_FOR


(*VACUUM PUMP*)
(*************************************************************************************************)


(*INK*)
(*************************************************************************************************)
FOR iL_Counter := 1 TO iCIk_NB_HEADERTANK DO
  fb_FillInkVarnish[iL_Counter].cI_Conf           := sC_Config_I.cC_CONF_INK_SUPPLY_UNIT;

  fb_Headertank[iL_Counter].bI_HeadertankExist    := bCIk_HEADERTANK_EXIST[iL_Counter];

  (*Messaging*)
  (*Config FB_HEADERTANK_UNIT*)
  fb_Headertank[iL_Counter].pC_MsgInterface       := ADR(sAdsIkHeaderTank[iL_Counter].sO_Message);
  fb_Headertank[iL_Counter].iC_BlockId            := eIk_BLK_HEADERTANK;
  fb_Headertank[iL_Counter].Init();

  (*Config FB_INK_SUPPLY_UNIT*)
  (*Only dummy, messaging is now handled by fb_Headertank*)
  fb_FillInkVarnish[iL_Counter].pC_MsgInterface   := ADR(sAdsIkDummy[1].sO_Message);  (*Only dummy, messages are not used in this FB*)
  fb_FillInkVarnish[iL_Counter].iC_BlockId        := 0;                               (*Messages are not used in this FB*)
  fb_FillInkVarnish[iL_Counter].Init();

  (*Circulation ink controller*)
  iSystemCmd.registerForSleepUpdate(iObserver:=fb_CirculationInk[iL_Counter]);
  
  fb_CirculationInk[iL_Counter].iPurgeController := fb_PurgeController[iCIk_MAP_HEADERTANK_PURGE_CONTR[iL_Counter]];
  fb_CirculationInk[iL_Counter].iMencController  := fb_MeniscusMencContr[iCIk_MAP_HEADERTANK_MENC_STA[iL_Counter]];
  fb_CirculationInk[iL_Counter].pName            := sC_Config_I.aC_HEADERTANK_NAME_DETAIL[iL_Counter];
END_FOR


(* STORAGE TANK *)
(**********************************************************************************)
FOR iL_Counter := 1 TO iCIk_NB_INKSTORAGE_TANK DO
  (*Messaging*)
  (*Config FB_STORAGETANK_UNIT*)
  fb_Storagetank[iL_Counter].pC_MsgInterface       := ADR(sAdsIkDummy[1].sO_Message);  (*ADR(sAdsIkInkStorageTank[iL_Counter].sO_Message);*)
  fb_Storagetank[iL_Counter].iC_BlockId            := eIk_BLK_INKSTORAGE_TANK;
  fb_Storagetank[iL_Counter].Init();

  (*Messaging*)
  sL_MsgConfigStorage[iL_Counter].bI_Enable       := TRUE;
  sL_MsgConfigStorage[iL_Counter].pI_FbMsgHandler := ADR(fB_BalanceMsgHandler[iL_Counter]);

  fB_BalanceMsgHandler[iL_Counter].pI_MsgQueue    := ADR(fB_MsgQueueStorage[iL_Counter]);

  fB_MsgQueueStorage[iL_Counter].pI_MsgInterface  := ADR(sAdsIkInkStorageTank[iL_Counter].sO_Message);
  fB_MsgQueueStorage[iL_Counter].cI_MaxElement    := 5;

  FOR iL_Counter2 := 1 TO iCIk_NB_BALANCE_MSG DO
    fB_BalanceMsg[iL_Counter, iL_Counter2].pI_MsgConfig   := ADR(sL_MsgConfigStorage[iL_Counter]);
    fB_BalanceMsg[iL_Counter, iL_Counter2].iI_MsgLocation := iL_Counter;
  END_FOR;

  fB_BalanceMsg[iL_Counter,  1].iI_MsgNumber      := eCIk_STOR_BAL_SEND;
  fB_BalanceMsg[iL_Counter,  2].iI_MsgNumber      := eCIk_STOR_BAL_RECEIVE;
  fB_BalanceMsg[iL_Counter,  3].iI_MsgNumber      := eCIk_STOR_BAL_MOTION;
  fB_BalanceMsg[iL_Counter,  4].iI_MsgNumber      := eCIk_STOR_BAL_NOCONNECT;
  fb_BalanceMsg[iL_Counter,  5].iI_MsgNumber      := eCIk_STOR_BAL_BUFFERFULL;
  fb_BalanceMsg[iL_Counter,  6].iI_MsgNumber      := eCIk_STOR_BAL_FRAMEFAULT;
  fb_BalanceMsg[iL_Counter,  7].iI_MsgNumber      := eCIk_STOR_BAL_OVERRUN;
  fb_BalanceMsg[iL_Counter,  8].iI_MsgNumber      := eCIk_STOR_LVL_WARNING;
  fb_BalanceMsg[iL_Counter,  9].iI_MsgNumber      := eCIk_STOR_LVL_ERROR;
  fb_BalanceMsg[iL_Counter, 10].iI_MsgNumber      := eCIk_STOR_TANK_MISSING;
  fb_BalanceMsg[iL_Counter, 11].iI_MsgNumber      := eCIk_STOR_TANK_MIXER_NOT_WORKING;
  fb_BalanceMsg[iL_Counter, 12].iI_MsgNumber      := eCIk_STOR_LVL_INFO;
  fb_BalanceMsg[iL_Counter, 13].iI_MsgNumber      := eCIk_STOR_SCAN_NEED;
  fb_BalanceMsg[iL_Counter, 14].iI_MsgNumber      := eCIk_STOR_SCAN_FALSE;
  fb_BalanceMsg[iL_Counter, 15].iI_MsgNumber      := eCIk_STOR_HT_ASSIGNMENT;
END_FOR;


(* BALANCE *)
(*************************************************************************************************)
(* -------------- init of the channels -------------------- *)
FOR iL_Counter := 1 TO iCIk_NB_INKBALANCE DO
  fb_Balance[iL_Counter].pI_BalanceOffset := ADR(fL_BalanceOffset[iL_Counter]);

  fb_BalanceLink.pI_ZeroPointerErr                 := ADR(nConvError);
  fb_BalanceLink.iI_UsedBalanceMux                 := iCIk_NB_BALANCE_MUX;
  fb_BalanceLink.bI_ZS_SelectedChannel[iL_Counter] := FALSE;
  fb_BalanceLink.bI_CS_SelectedChannel[iL_Counter] := FALSE;

  fb_BalanceLink( cI_MapBalanceBalanceMux     := cCIk_MAP_BALANCE_BALANCE_MUX
                , cI_MapBalanceBalanceChannel := cCIk_MAP_BALANCE_BALANCE_CHANNEL);
  
END_FOR;


  
(*************************************************************************************************)
(*ADS blocks mapping*)
(*************************************************************************************************)

(*Recipe read/write*)
(*************************************************************************************************)
IF cL_State = cL_INIT_PRG THEN
  pFbRecipeMngr := PRG_SYSTEMBASE.registerRecipe(
    aI_RecipePath           := CONCAT(aC_PlcConfigPath, aC_PlcRecipeSubPath),
    aI_RecipeDefinitionName := sC_Ads_Info.aType  (*is set in Mapping*)
  );
 
  (* -- BlockId saving ----------------------------------------------------------------------------*)
  PRG_SYSTEMBASE.fbBlockIdSave.registerModule(
    aI_StoragePath := CONCAT(aC_PlcConfigPath, aC_PlcBlockIdSubPath),
    pI_Ads_Info    := ADR(sC_Ads_Info)
  );
END_IF


(********************************* END OF ACTION *************************************************)
END_ACTION

ACTION Mapping:
(*************************************************************************************************)
(*ADS blocks mapping definition*)
(*************************************************************************************************)
(*mapping of each block with his parents, unique type and index*)

(*purge controller*)
FOR iL_Counter := 1 TO iCIk_NB_PURGE_CONTR DO
  IF bCIk_PURGE_CONTR_EXIST[iL_Counter] THEN
    (*purge controller -> root*)
		sL_BLK_PURGE_CONTR[iL_Counter].iPMaps[1]    := FC_ADD_MAP(eSys_BLK_ROOT, 1);
  END_IF;
END_FOR;

(*purge group*)
FOR iL_Counter := 1 TO iCIk_NB_PURGE_GROUP DO
  IF bCIk_PURGE_GROUP_EXIST[iL_Counter] THEN
    (*purge group -> purge controller*)
    sL_BLK_PURGE_GROUP[iL_Counter].iPMaps[1]      := FC_ADD_MAP(eIk_BLK_PURGE_CONTROLLER, cCIk_MAP_PURGE_GROUP_CONTR[iL_Counter]);
  END_IF;
END_FOR;

(*dgas*)
FOR iL_Counter := 1 TO iCIk_NB_DGAS DO
  (*dgas -> root*)
  sL_BLK_DGAS[iL_Counter].iPMaps[1]             := FC_ADD_MAP(eSys_BLK_ROOT, 1);
  (*dgas -> purge*)
(*sL_BLK_DGAS[iL_Counter].iPMaps[2]             := FC_ADD_MAP(eIk_BLK_PURGE_CONTROLLER, 1);
  sL_BLK_DGAS[iL_Counter].iPMaps[3]             := FC_ADD_MAP(eIk_BLK_PURGE_CONTROLLER, 2);*)
END_FOR;

(*menc*)
FOR iL_Counter := 1 TO iCIk_NB_MENC DO
  (*main menc -> root*)
  sL_BLK_MENC[iL_Counter].iPMaps[1]             := FC_ADD_MAP(eSys_BLK_ROOT, 1);
END_FOR;
FOR iL_Counter := 1 TO iCIk_NB_SUB_MENC DO
  (*sub menc -> menc*)
  sL_BLK_MENC[iCIk_NB_MENC + iL_Counter].iPMaps[1] := FC_ADD_MAP(eIk_BLK_MENC, iCIk_MAP_SUB_MENC_MAIN_MENC[iL_Counter]);
  (*sub menc -> header tank group*)
  sL_BLK_MENC[iCIk_NB_MENC + iL_Counter].iPMaps[2] := FC_ADD_MAP(eIk_BLK_HEADERTANK_GROUP, iCIk_MAP_SUB_MENC_HTG[iL_Counter]);
END_FOR;

(*ink storage tank*)
FOR iL_Counter := 1 TO iCIk_NB_INKSTORAGE_TANK DO
  IF bCIk_INKSTORAGE_TANK_EXIST[iL_Counter] THEN
    (*ink storage tank -> root*)
    sL_BLK_INKSTORAGE_TANK[iL_Counter].iPMaps[1] := FC_ADD_MAP(eSys_BLK_ROOT, 1);
  END_IF;
END_FOR;

(*header tank group*)
FOR iL_Counter := 1 TO iCIk_NB_HEADERTANK_GROUP DO
  (*header tank group -> storage tank*)
  sL_BLK_HEADERTANK_GROUP[iL_Counter].iPMaps[1]   := FC_ADD_MAP(eIk_BLK_INKSTORAGE_TANK, 1);
  sL_BLK_HEADERTANK_GROUP[iL_Counter].iPMaps[2]   := FC_ADD_MAP(eIk_BLK_INKSTORAGE_TANK, 2);
END_FOR;

(*header tank*)
FOR iL_Counter := 1 TO iCIk_NB_HEADERTANK DO
  IF bCIk_HEADERTANK_EXIST[iL_Counter] THEN
    (*header tank -> storage tank*)
    sL_BLK_HEADERTANK[iL_Counter].iPMaps[1]       := FC_ADD_MAP(eIk_BLK_INKSTORAGE_TANK, 1);
    sL_BLK_HEADERTANK[iL_Counter].iPMaps[2]       := FC_ADD_MAP(eIk_BLK_INKSTORAGE_TANK, 2);

    (*header tank -> meniscus*)
    sL_BLK_HEADERTANK[iL_Counter].iPMaps[3]       := FC_ADD_MAP(eIk_BLK_MENC, iCIk_MAP_HEADERTANK_MENC_STA[iL_Counter]);

    (*header tank -> header tank group*)
    sL_BLK_HEADERTANK[iL_Counter].iPMaps[4]       := FC_ADD_MAP(eIk_BLK_HEADERTANK_GROUP, iCIk_MAP_HEADERTANK_HT_GROUP[iL_Counter]);
  END_IF;
END_FOR;

(*heater*)
FOR iL_Counter := 1 TO iCIk_NB_TEMP_CONTR DO
  (*heater -> root*)
  sL_BLK_HEATER[iL_Counter].iPMaps[1]           := FC_ADD_MAP(eSys_BLK_ROOT, 1);
  (*heater -> group*)
  sL_BLK_HEATER[iL_Counter].iPMaps[2]           := FC_ADD_MAP(ePr_BLK_PG, iCIk_MAP_TEMP_PG[iL_Counter]);
END_FOR;


(*ADS blocks configuration & information*)
(*************************************************************************************************)
sC_Ads_Info.bReady   := FALSE;
sC_Ads_Info.aType    := 'PRG_INK';
sC_Ads_Info.iVersion := 010000;        (*1.0.0*)
sC_Ads_Info.iType    := eMOD_INK;

sMappingInfo.init(lModId:=TO_UINT(eMOD_INK)); 
sMappingInfo.addBlkAry( iAdsBlockType := TO_UINT(eIk_BLK_PURGE_CONTROLLER), aAdsBlockName := 'sAdsIkPurgeController', iAdsBlockVersion:= INT_TO_UINT(sAdsIkPurgeController[1].iO_Version), iNbrBlocks := SIZEOF(sL_BLK_PURGE_CONTR)     / SIZEOF(sL_BLK_PURGE_CONTR[1]),     pBlockArray := ADR(sL_BLK_PURGE_CONTR));
sMappingInfo.addBlkAry( iAdsBlockType := TO_UINT(eIk_BLK_PURGE_GROUP),      aAdsBlockName := 'sAdsIkPurgeGroup',      iAdsBlockVersion:= INT_TO_UINT(sAdsIkPurgeGroup[1].iO_Version),      iNbrBlocks := SIZEOF(sL_BLK_PURGE_GROUP)     / SIZEOF(sL_BLK_PURGE_GROUP[1]),     pBlockArray := ADR(sL_BLK_PURGE_GROUP));
sMappingInfo.addBlkAry( iAdsBlockType := TO_UINT(eIk_BLK_DGAS),             aAdsBlockName := 'sAdsIkDgas',            iAdsBlockVersion:= INT_TO_UINT(sAdsIkDgas[1].iO_Version),            iNbrBlocks := SIZEOF(sL_BLK_DGAS)            / SIZEOF(sL_BLK_DGAS[1]),            pBlockArray := ADR(sL_BLK_DGAS));
sMappingInfo.addBlkAry( iAdsBlockType := TO_UINT(eIk_BLK_MENC),             aAdsBlockName := 'sAdsIkMenc',            iAdsBlockVersion:= INT_TO_UINT(sAdsIkMenc[1].iO_Version),            iNbrBlocks := SIZEOF(sL_BLK_MENC)            / SIZEOF(sL_BLK_MENC[1]),            pBlockArray := ADR(sL_BLK_MENC));
sMappingInfo.addBlkAry( iAdsBlockType := TO_UINT(eIk_BLK_HEADERTANK_GROUP), aAdsBlockName := 'sAdsIkHeaderTankGroup', iAdsBlockVersion:= INT_TO_UINT(sAdsIkHeaderTankGroup[1].iO_Version), iNbrBlocks := SIZEOF(sL_BLK_HEADERTANK_GROUP)/ SIZEOF(sL_BLK_HEADERTANK_GROUP[1]),pBlockArray := ADR(sL_BLK_HEADERTANK_GROUP));
sMappingInfo.addBlkAry( iAdsBlockType := TO_UINT(eIk_BLK_HEADERTANK),       aAdsBlockName := 'sAdsIkHeaderTank',      iAdsBlockVersion:= INT_TO_UINT(sAdsIkHeaderTank[1].iO_Version),      iNbrBlocks := SIZEOF(sL_BLK_HEADERTANK)      / SIZEOF(sL_BLK_HEADERTANK[1]),      pBlockArray := ADR(sL_BLK_HEADERTANK));
sMappingInfo.addBlkAry( iAdsBlockType := TO_UINT(eIk_BLK_INKSTORAGE_TANK),  aAdsBlockName := 'sAdsIkInkStorageTank',  iAdsBlockVersion:= INT_TO_UINT(sAdsIkInkStorageTank[1].iO_Version),  iNbrBlocks := SIZEOF(sL_BLK_INKSTORAGE_TANK) / SIZEOF(sL_BLK_INKSTORAGE_TANK[1]), pBlockArray := ADR(sL_BLK_INKSTORAGE_TANK));
sMappingInfo.addBlkAry( iAdsBlockType := TO_UINT(eIk_BLK_INKPUMP),          aAdsBlockName := 'sAdsIkInkPump',         iAdsBlockVersion:= INT_TO_UINT(sAdsIkInkPump[1].iO_Version),         iNbrBlocks := SIZEOF(sL_BLK_INKPUMP)         / SIZEOF(sL_BLK_INKPUMP[1]),         pBlockArray := ADR(sL_BLK_INKPUMP));
sMappingInfo.addBlkAry( iAdsBlockType := TO_UINT(eIk_BLK_HEATER),           aAdsBlockName := 'sAdsIkHeater',          iAdsBlockVersion:= INT_TO_UINT(sAdsIkHeater[1].iO_Version),          iNbrBlocks := SIZEOF(sL_BLK_HEATER)          / SIZEOF(sL_BLK_HEATER[1]),          pBlockArray := ADR(sL_BLK_HEATER));
sMappingInfo.bReady := TRUE;

// Register module
ISystemBase.regModule( pAdsInfo := ADR(sC_Ads_Info)
                     , pMapInfo := ADR(sMappingInfo) );

(********************************* END OF ACTION *************************************************)
END_ACTION

ACTION RemVar:
(*************************************************************************************************)
(********************************* READING REMANENT VARIABLES ************************************)
(*************************************************************************************************)
IF bL_RemVar_Init THEN

  (*load initial values if pattern was invalid*)
  IF sR_RemVar_I.aL_Pattern <> 16#ABCD THEN

    (*initial very boot values of project*)
    sR_RemVar_I.aL_Pattern := 16#ABCD;

    (*TODO add boot/config values*)

    (*DEGASSING*)
    (*************************************************************************************************)
    FOR iL_Counter := 1 TO iCIk_NB_DGAS DO
      sAdsIkDgas[iL_Counter].sI_PressSet.fI_Val             := -400;   (*mbar*)
    END_FOR;


    (*MENISCUS*)
    (*************************************************************************************************)
    (*Main*)
    sAdsIkMenc[1].sI_PressSet.fI_Val                        := sC_Config_I.fL_MENC1_PRESS_INITVAL;       (*mbar*)
    (*Sub*)
    sAdsIkMenc[2].sI_PressSet.fI_Val                        := sC_Config_I.fL_SUB_MENC1_PRESS_INITVAL;   (*mbar*)
    sAdsIkMenc[3].sI_PressSet.fI_Val                        := sC_Config_I.fL_SUB_MENC2_PRESS_INITVAL;   (*mbar*)

    (*Init rem var*)
    FOR iL_CounterMenc := 1 TO iCIk_NB_MENC DO
      fb_MeniscusMencContr[iL_CounterMenc].mInitRemVar( IfConvAdsTtLocal := sC_Config_I.fL_MENC_CONV_ADS_TO_LCL
                                                      , IfPressSetMin    := sC_Config_I.fL_MENC_PRESS_SET_MIN
                                                      , IfPressSetMax    := sC_Config_I.fL_MENC_PRESS_SET_MAX
                                                      , IfPressActMin    := sC_Config_I.fL_MENC_PRESS_ACT_MIN
                                                      , IfPressActMax    := sC_Config_I.fL_MENC_PRESS_ACT_MAX
                                                      , IfTolSmall       := sC_Config_I.fL_MENC_TOL_SMALL
                                                      , IfTolBig         := sC_Config_I.fL_MENC_TOL_BIG);
    END_FOR;
    FOR iL_CounterSubMenc := 1 TO iCIk_NB_SUB_MENC DO
      (*Special for sub men white pos*)
      IF sC_Config_I.aC_SUB_MENC_NAME_DETAIL[iL_CounterSubMenc] = 'Sub White pos' THEN
        fb_MeniscusMencContr[iCIk_NB_MENC + iL_CounterSubMenc].mInitRemVar( IfConvAdsTtLocal := sC_Config_I.fL_SUB_MENC_CONV_ADS_TO_LCL
                                                                          , IfPressSetMin    :=  -2.0
                                                                          , IfPressSetMax    := 120.0
                                                                          , IfPressActMin    :=  -2.0
                                                                          , IfPressActMax    := 120.0
                                                                          , IfTolSmall       := sC_Config_I.fL_SUB_MENC_TOL_SMALL
                                                                          , IfTolBig         := sC_Config_I.fL_SUB_MENC_TOL_BIG);
      ELSE
        fb_MeniscusMencContr[iCIk_NB_MENC + iL_CounterSubMenc].mInitRemVar( IfConvAdsTtLocal := sC_Config_I.fL_SUB_MENC_CONV_ADS_TO_LCL
                                                                          , IfPressSetMin    := sC_Config_I.fL_SUB_MENC_PRESS_SET_MIN
                                                                          , IfPressSetMax    := sC_Config_I.fL_SUB_MENC_PRESS_SET_MAX
                                                                          , IfPressActMin    := sC_Config_I.fL_SUB_MENC_PRESS_ACT_MIN
                                                                          , IfPressActMax    := sC_Config_I.fL_SUB_MENC_PRESS_ACT_MAX
                                                                          , IfTolSmall       := sC_Config_I.fL_SUB_MENC_TOL_SMALL
                                                                          , IfTolBig         := sC_Config_I.fL_SUB_MENC_TOL_BIG);
			END_IF
    END_FOR;
    
    (*INK*)
    (*************************************************************************************************)
    (*varnish*)
    FOR iL_Counter:= 1 TO iCIk_NB_HEADERTANK DO
      sAdsIkHeaderTank[iL_Counter].bI_FillModeAuto          := TRUE;
      sAdsIkHeaderTank[iL_Counter].bI_EnableRamp            := FALSE;
    END_FOR

    
    (*MAINTENANCE*)
    (*************************************************************************************************)
    (*VISU SETTINGS*)
		wIDp_MinSpeedFillInkPumpVarnish                         := 10;     (*%*)
		wIDp_MaxSpeedFillInkPumpVarnish                         := 100;    (*%*)
		wIDP_AnalogMinDigitVarnish                              := 0;
		wIDP_AnalogMaxDigitVarnish                              := 16383;

    lL_TimeReturnFlow                                       := 90;     (*s*)
    lL_TimeBlowOut                                          := 130;    (*s*)
    lL_TimeEmptyCleaner                                     := 60;     (*s*)
    lL_TimeWarnExchange                                     := 6;      (*h*)

    
    (*TEMP*)
    (*************************************************************************************************)
    FOR iL_Counter := 1 TO iCIk_NB_TEMP_CONTR DO
      sAdsIkHeater[iL_Counter].sI_HeaterSet.fI_Val          := 50;    (*°C*)
    END_FOR

    
    (*PURGE*)
    (*************************************************************************************************)
    sAdsIkPurgeController[1].bI_Enable                      := TRUE;

    
		(*BALANCE*)
		(*************************************************************************************************)
		bI_EnableBalanceLink                                            := TRUE;
		fI_CorrectionValue                                              := 1.00;
		iI_RefreshRate                                                  := 2000;   (*ms*)
		FOR iL_Counter := 1 TO iCIk_NB_INKSTORAGE_TANK DO
			sAdsIkInkStorageTank[iL_Counter].sI_EnableBalance.bI_Command  := TRUE;

			sAdsIkInkStorageTank[iL_Counter].sI_InkDensitySet.fI_Val      := 1.07;
			sAdsIkInkStorageTank[iL_Counter].sI_CorrectionValue.fI_Val    := 1.00;
			sAdsIkInkStorageTank[iL_Counter].fO_StorageTankSize           := 25.0;   (*l*)

			sAdsIkInkStorageTank[iL_Counter].sI_WarningLevelSet.fI_Val    := 4.0;
			sAdsIkInkStorageTank[iL_Counter].sI_ErrorlevelSet.fI_Val      := 3.0;
			sAdsIkInkStorageTank[iL_Counter].sI_MaintenanceTimeout.lI_Val := 5000;

      (*Varnish parameter*)
      sAdsIkInkStorageTank[iL_Counter].sI_InkParameter.aWaveform           := 'waveform.wav';
      sAdsIkInkStorageTank[iL_Counter].sI_InkParameter.sTemperature.fI_Val := 35.0;
      sAdsIkInkStorageTank[iL_Counter].sI_InkParameter.sMeniscus.fI_Val    := -24.5;
      sAdsIkInkStorageTank[iL_Counter].sI_InkParameter.sDensity.fI_Val     := 1.0;
      sAdsIkInkStorageTank[iL_Counter].sI_InkParameter.sViscosity.fI_Val   := 100.0;
		END_FOR

		FOR iL_Counter := 1 TO iCIk_NB_INKBALANCE DO
      fL_BalanceOffset[iL_Counter]                                  := 0;

			sAdsIkInkStorageTank[iL_Counter].aI_CalibrateFrameText1       := 'aaaaaaaa';
			sAdsIkInkStorageTank[iL_Counter].aI_CalibrateFrameText2       := 'bbbbbbbb';
		END_FOR;
		sAdsIkInkStorageTank[1].aI_CalibrateFrameText1                  := '4D5A2406';
		sAdsIkInkStorageTank[1].aI_CalibrateFrameText2                  := '399128E6';
		sAdsIkInkStorageTank[2].aI_CalibrateFrameText1                  := '4D5426F9';
		sAdsIkInkStorageTank[2].aI_CalibrateFrameText2                  := '3991CD5A';
		sAdsIkInkStorageTank[3].aI_CalibrateFrameText1                  := 'aaaaaaaa';
		sAdsIkInkStorageTank[3].aI_CalibrateFrameText2                  := 'bbbbbbbb';

    (*Recipe: load and write*)
    IF pFbRecipeMngr <> 0 THEN
      pFbRecipeMngr^.mWriteRecipe('');
      PRG_MACHINE.bI_RecipeValuesLoadedInk := TRUE;
    END_IF

  ELSE

    sR_RemVar_I.aL_Pattern := sR_RemVar_I.aL_Pattern;  (*TODO remove dummy code*)

    (*DEGASSING*)
    (*************************************************************************************************)
    sAdsIkDgas[1].bI_Enable             := sR_RemVar_I.lR_DgasEnable;
    sAdsIkDgas[1].sI_PressSet.fI_Val    := (sR_RemVar_I.fR_DgasPressStpt * sC_Config_I.fL_DGAS1_CONV_ADS_TO_LCL);

    bIDp_EnableMainDgasValve            := sR_RemVar_I.lR_DgasEnableMainValve;
    sC_Config_I.lL_DGAS_TIME_ERROR      := sR_RemVar_I.lR_DgasTimeError;


    (*MENISCUS*)
    (*************************************************************************************************)
    FOR iL_Counter := 1 TO iCIk_NB_MENC DO
      sAdsIkMenc[iL_Counter].bI_Enable                         := sR_RemVar_I.lR_MencEnable   [iL_Counter];
      sAdsIkMenc[iL_Counter].sI_PressSet.fI_Val                := sR_RemVar_I.fR_MencPressStpt[iL_Counter];
    END_FOR;

    sC_Config_I.wL_MENC_TIME_ERROR                             := sR_RemVar_I.wR_MencTimeError;
    sC_Config_I.wL_SUB_MENC_TIME_ERROR                         := sR_RemVar_I.wR_SubMencTimeError;


    (*SUB MENISCUS*)
    (*************************************************************************************************)
    (*Sub meniscus starts behind the meniscus*)
    FOR iL_Counter := 1 TO iCIk_NB_SUB_MENC DO
      sAdsIkMenc[iCIk_NB_MENC + iL_Counter].bI_Enable          := sR_RemVar_I.lR_SubMencEnable        [iL_Counter];
      sAdsIkMenc[iCIk_NB_MENC + iL_Counter].sI_PressSet.fI_Val := sR_RemVar_I.fR_SubMencPressStpt     [iL_Counter];
    END_FOR;


    (*INK*)
    (*************************************************************************************************)
    (*varnish*)
    FOR iL_Counter := 1 TO iCIk_NB_HEADERTANK DO
      sAdsIkHeaderTank[iL_Counter].sI_StoragetankAssignment.lI_Val    := sR_RemVar_I.lR_StoragetankAssignment[iL_Counter];
      sAdsIkHeaderTank[iL_Counter].sO_ActStoragetankAssignment.lI_Val := sR_RemVar_I.lR_ActStoragetankAssignment[iL_Counter];
      
      sAdsIkHeaderTank[iL_Counter].bI_EnableFillInk       := sR_RemVar_I.bI_EnableFillInk[iL_Counter];
      sAdsIkHeaderTank[iL_Counter].bI_FillModeAuto        := sR_RemVar_I.bI_FillModeAuto[iL_Counter];
      sAdsIkHeaderTank[iL_Counter].bI_EnableUnFillInk     := sR_RemVar_I.bI_EnableUnFillInk[iL_Counter];
      sAdsIkHeaderTank[iL_Counter].bI_UnFillModeAuto      := sR_RemVar_I.bI_UnFillModeAuto[iL_Counter];

      sAdsIkInkPump[iL_Counter].sI_InkPumpSpeedSet.lI_Val := WORD_TO_DINT(sR_RemVar_I.wR_StptSpeedFillInkPumpVarnishPercent[iL_Counter]);

      fb_Headertank[iL_Counter].StateHeadertank           := sR_RemVar_I.eR_StateHeadertank[iL_Counter];
    END_FOR

		wIDp_MinSpeedFillInkPumpVarnish								:= sR_RemVar_I.wR_MinSpeedFillInkPumpVarnish;
		wIDp_MaxSpeedFillInkPumpVarnish								:= sR_RemVar_I.wR_MaxSpeedFillInkPumpVarnish;
		wIDP_AnalogMinDigitVarnish 										:= sR_RemVar_I.wR_AnalogMinDigitVarnish;
		wIDP_AnalogMaxDigitVarnish 										:= sR_RemVar_I.wR_AnalogMaxDigitVarnish;
		wIDp_PumpTimeOffDelayVarnish									:= sR_RemVar_I.wR_PumpTimeOffDelayVarnish;

    lL_TimeReturnFlow                             := sR_RemVar_I.lR_TimeReturnFlow;
    lL_TimeBlowOut                                := sR_RemVar_I.lR_TimeBlowOut;
    lL_TimeEmptyCleaner                           := sR_RemVar_I.lR_TimeEmptyCleaner;
    lL_TimeWarnExchange                           := sR_RemVar_I.lR_TimeWarnExchange;

    sC_Config_I.wC_INKPUMP_MAX_TIME               := sR_RemVar_I.wR_InkPumpMaxTime;
    sC_Config_I.wC_CLEANERPUMP_MAX_TIME           := sR_RemVar_I.wR_CleanerPumpMaxTime;

    
    (*TEMP*)
    (*************************************************************************************************)
    FOR iL_Counter :=1 TO iCIk_NB_TEMP_CONTR DO
      sAdsIkHeater[iL_Counter].bI_EnableHeater     := sR_RemVar_I.bI_EnableHeater  [iL_Counter];
      sAdsIkHeater[iL_Counter].sI_HeaterSet.fI_Val := sR_RemVar_I.sI_HeaterSetPoint[iL_Counter];
    END_FOR


    (*PURGE*)
    (*************************************************************************************************)
    FOR iL_Counter := 1 TO iCIk_NB_PURGE_CONTR DO
      sAdsIkPurgeController[iL_Counter].bI_Enable         := sR_RemVar_I.bR_PurgeControllerEnable[iL_Counter];
    END_FOR;

    FOR iL_Counter := 1 TO iCIk_NB_PURGE_GROUP DO
      sAdsIkPurgeGroup[iL_Counter].bI_EnablePurge         := sR_RemVar_I.bR_PurgeGroupEnable       [iL_Counter];
      sAdsIkPurgeGroup[iL_Counter].bI_EnableThroughNozzle := sR_RemVar_I.bR_PurgeGroupThroughNozzle[iL_Counter];
      sAdsIkPurgeGroup[iL_Counter].bI_EnableFlush         := sR_RemVar_I.bR_PurgeGroupFlush        [iL_Counter];
    END_FOR;


		(*BALANCE*)
		(*************************************************************************************************)
		bI_EnableBalanceLink    := sR_RemVar_I.bI_EnableBalanceLink;
		fI_CorrectionValue      := sR_RemVar_I.fI_CorrectionValue;
		iI_RefreshRate          := sR_RemVar_I.iI_RefreshRate;
		iI_MaintenanceTimeout   := sR_RemVar_I.iI_MaintenanceTimeout;

		FOR iL_Counter := 1 TO iCIk_NB_INKSTORAGE_TANK DO
			sAdsIkInkStorageTank[iL_Counter].bI_EnableStorageTank        := sR_RemVar_I.bI_EnableStorageTank[iL_Counter];
			sAdsIkInkStorageTank[iL_Counter].lO_InkColorId               := sR_RemVar_I.lO_InkColorId[iL_Counter];
			sAdsIkInkStorageTank[iL_Counter].fO_StorageTankSize          := sR_RemVar_I.fO_StorageTankSize[iL_Counter];
		END_FOR;

		FOR iL_Counter := 1 TO iCIk_NB_INKBALANCE DO
			sAdsIkInkStorageTank[iL_Counter].sI_EnableBalance.bI_Command := sR_RemVar_I.bI_EnableBalance[iL_Counter];
			sAdsIkInkStorageTank[iL_Counter].sI_InkDensitySet.fI_Val     := sR_RemVar_I.sI_InkDensitySet[iL_Counter];
			sAdsIkInkStorageTank[iL_Counter].sI_CorrectionValue.fI_Val   := sR_RemVar_I.sI_CorrectionValue[iL_Counter];
			sAdsIkInkStorageTank[iL_Counter].sI_WarningLevelSet.fI_Val   := sR_RemVar_I.sI_WarningLevelSet[iL_Counter];
			sAdsIkInkStorageTank[iL_Counter].sI_ErrorlevelSet.fI_Val     := sR_RemVar_I.sI_ErrorlevelSet[iL_Counter];

      (*Varnish parameter*)
      sAdsIkInkStorageTank[iL_Counter].sI_InkParameter.iScannerId          := sR_RemVar_I.lR_VarParamScannerId[iL_Counter];
      sAdsIkInkStorageTank[iL_Counter].sI_InkParameter.iIndex              := sR_RemVar_I.iR_VarParamIndex[iL_Counter];
      sAdsIkInkStorageTank[iL_Counter].sI_InkParameter.sTemperature.fI_Val := sR_RemVar_I.fR_VarParamTemp[iL_Counter];
      sAdsIkInkStorageTank[iL_Counter].sI_InkParameter.sMeniscus.fI_Val    := sR_RemVar_I.fR_VarParamMenc[iL_Counter];
      sAdsIkInkStorageTank[iL_Counter].sI_InkParameter.aWaveform           := sR_RemVar_I.aR_VarParamWaveform[iL_Counter];
      sAdsIkInkStorageTank[iL_Counter].sI_InkParameter.iTimer              := sR_RemVar_I.iR_VarParamTimer[iL_Counter];
      sAdsIkInkStorageTank[iL_Counter].sI_InkParameter.sDensity.fI_Val     := sR_RemVar_I.fR_VarParamDensity[iL_Counter];
      sAdsIkInkStorageTank[iL_Counter].sI_InkParameter.sViscosity.fI_Val   := sR_RemVar_I.fR_VarParamViscosity[iL_Counter];
      sAdsIkInkStorageTank[iL_Counter].sI_InkParameter.iColorId            := sR_RemVar_I.iR_VarParamColorId[iL_Counter];
      FOR iL_Counter2 := 1 TO 10 DO
        sAdsIkInkStorageTank[iL_Counter].sI_InkParameter.bCompatibility[iL_Counter2] := sR_RemVar_I.bR_VarParamCompatibility[iL_Counter, iL_Counter2];
      END_FOR;

			sAdsIkInkStorageTank[iL_Counter].aI_CalibrateFrameText1      := sR_RemVar_I.aI_CalibrateFrameText1[iL_Counter];
			sAdsIkInkStorageTank[iL_Counter].aI_CalibrateFrameText2      := sR_RemVar_I.aI_CalibrateFrameText2[iL_Counter];

      fL_BalanceOffset[iL_Counter] := sR_RemVar_I.fR_BalanceOffset[iL_Counter];
		END_FOR;

  END_IF


  bL_RemVar_Init := FALSE;



(*************************************************************************************************)
(********************************* WRITING REMANENT VARIABLES ************************************)
(*************************************************************************************************)
ELSE

(*GENERAL*)
(*************************************************************************************************)
  sR_RemVar_I.aL_Pattern := 16#ABCD;

(*DEGASSING*)
(*************************************************************************************************)
  sR_RemVar_I.lR_DgasEnable           := sAdsIkDgas[1].bI_Enable;
  sR_RemVar_I.fR_DgasPressStpt        := sAdsIkDgas[1].sI_PressSet.fI_Val;

  sR_RemVar_I.lR_DgasEnableMainValve  := bIDp_EnableMainDgasValve;
  sR_RemVar_I.lR_DgasTimeError        := sC_Config_I.lL_DGAS_TIME_ERROR;

(*MENISCUS*)
(*************************************************************************************************)
  FOR iL_Counter := 1 TO iCIk_NB_MENC DO
    sR_RemVar_I.fR_MencPressStpt[iL_Counter]      := sAdsIkMenc[iL_Counter].sI_PressSet.fI_Val;
    sR_RemVar_I.lR_MencEnable   [iL_Counter]      := sAdsIkMenc[iL_Counter].bI_Enable;
  END_FOR;

  sR_RemVar_I.wR_MencTimeError                    := sC_Config_I.wL_MENC_TIME_ERROR;
  sR_RemVar_I.wR_SubMencTimeError                 := sC_Config_I.wL_SUB_MENC_TIME_ERROR;

(*SUB MENISCUS*)
(*************************************************************************************************)
  (*Sub meniscus starts behind the meniscus*)
  FOR iL_Counter := 1 TO iCIk_NB_SUB_MENC DO
    sR_RemVar_I.fR_SubMencPressStpt     [iL_Counter] := sAdsIkMenc[iCIk_NB_MENC + iL_Counter].sI_PressSet.fI_Val;
    sR_RemVar_I.lR_SubMencEnable        [iL_Counter] := sAdsIkMenc[iCIk_NB_MENC + iL_Counter].bI_Enable;
  END_FOR;

(*PURGE - GLOBAL*)
(*************************************************************************************************)
  FOR iL_Counter := 1 TO iCIk_NB_PURGE_CONTR DO
    sR_RemVar_I.bR_PurgeControllerEnable  [iL_Counter] := sAdsIkPurgeController[iL_Counter].bI_Enable;
  END_FOR;

  FOR iL_Counter := 1 TO iCIk_NB_PURGE_GROUP DO
    sR_RemVar_I.bR_PurgeGroupEnable       [iL_Counter] := sAdsIkPurgeGroup[iL_Counter].bI_EnablePurge;
    sR_RemVar_I.bR_PurgeGroupThroughNozzle[iL_Counter] := sAdsIkPurgeGroup[iL_Counter].bI_EnableThroughNozzle;
    sR_RemVar_I.bR_PurgeGroupFlush        [iL_Counter] := sAdsIkPurgeGroup[iL_Counter].bI_EnableFlush;
  END_FOR;


(*INK*)
(*************************************************************************************************)
  (*varnish*)
  FOR iL_Counter:= 1 TO iCIk_NB_HEADERTANK DO
    sR_RemVar_I.lR_StoragetankAssignment   [iL_Counter]           := sAdsIkHeaderTank[iL_Counter].sI_StoragetankAssignment.lI_Val;
    sR_RemVar_I.lR_ActStoragetankAssignment[iL_Counter]           := sAdsIkHeaderTank[iL_Counter].sO_ActStoragetankAssignment.lI_Val;
      
    sR_RemVar_I.bI_EnableFillInk  [iL_Counter]                    := sAdsIkHeaderTank[iL_Counter].bI_EnableFillInk;
    sR_RemVar_I.bI_FillModeAuto   [iL_Counter]                    := sAdsIkHeaderTank[iL_Counter].bI_FillModeAuto;
    sR_RemVar_I.bI_EnableUnFillInk[iL_Counter]                    := sAdsIkHeaderTank[iL_Counter].bI_EnableUnFillInk;
    sR_RemVar_I.bI_UnFillModeAuto [iL_Counter]                    := sAdsIkHeaderTank[iL_Counter].bI_UnFillModeAuto;

    sR_RemVar_I.wR_StptSpeedFillInkPumpVarnishPercent[iL_Counter] := DINT_TO_WORD(sAdsIkInkPump[iL_Counter].sI_InkPumpSpeedSet.lI_Val);
    
    sR_RemVar_I.eR_StateHeadertank[iL_Counter]                    := fb_Headertank[iL_Counter].StateHeadertank;
  END_FOR

	sR_RemVar_I.wR_MinSpeedFillInkPumpVarnish 				:= wIDp_MinSpeedFillInkPumpVarnish;
	sR_RemVar_I.wR_MaxSpeedFillInkPumpVarnish					:= wIDp_MaxSpeedFillInkPumpVarnish;
	sR_RemVar_I.wR_AnalogMinDigitVarnish 							:= wIDP_AnalogMinDigitVarnish;
	sR_RemVar_I.wR_AnalogMaxDigitVarnish 							:= wIDP_AnalogMaxDigitVarnish;
	sR_RemVar_I.wR_PumpTimeOffDelayVarnish 						:= wIDp_PumpTimeOffDelayVarnish;

  sR_RemVar_I.lR_TimeReturnFlow                     := lL_TimeReturnFlow;
  sR_RemVar_I.lR_TimeBlowOut                        := lL_TimeBlowOut;
  sR_RemVar_I.lR_TimeEmptyCleaner                   := lL_TimeEmptyCleaner;
  sR_RemVar_I.lR_TimeWarnExchange                   := lL_TimeWarnExchange;

  sR_RemVar_I.wR_InkPumpMaxTime                     := sC_Config_I.wC_INKPUMP_MAX_TIME;
  sR_RemVar_I.wR_CleanerPumpMaxTime                 := sC_Config_I.wC_CLEANERPUMP_MAX_TIME;


(*RAMPE*)
(*************************************************************************************************)


(*TEMP*)
(*************************************************************************************************)
  FOR iL_Counter := 1 TO iCIk_NB_TEMP_CONTR DO
    sR_RemVar_I.bI_EnableHeater  [iL_Counter] := sAdsIkHeater[iL_Counter].bI_EnableHeater;
    sR_RemVar_I.sI_HeaterSetPoint[iL_Counter] := sAdsIkHeater[iL_Counter].sI_HeaterSet.fI_Val;
  END_FOR

  
(*INKSTORAGE_TANK*)
(*************************************************************************************************)
  FOR iL_Counter := 1 TO iCIk_NB_INKSTORAGE_TANK DO
    sR_RemVar_I.bI_EnableStorageTank[iL_Counter] := sAdsIkInkStorageTank[iL_Counter].bI_EnableStorageTank;
    sR_RemVar_I.lO_InkColorId[iL_Counter]        := sAdsIkInkStorageTank[iL_Counter].lO_InkColorId;
    sR_RemVar_I.fO_StorageTankSize[iL_Counter]   := sAdsIkInkStorageTank[iL_Counter].fO_StorageTankSize;
  END_FOR;

	(*BALANCE*)
	sR_RemVar_I.bI_EnableBalanceLink  := bI_EnableBalanceLink;
	sR_RemVar_I.fI_CorrectionValue    := fI_CorrectionValue;
	sR_RemVar_I.iI_RefreshRate        := iI_RefreshRate;
	sR_RemVar_I.iI_MaintenanceTimeout := iI_MaintenanceTimeout;

  FOR iL_Counter := 1 TO iCIk_NB_INKBALANCE DO
    sR_RemVar_I.bI_EnableBalance    [iL_Counter]   := sAdsIkInkStorageTank[iL_Counter].sI_EnableBalance.bI_Command;
    sR_RemVar_I.sI_InkDensitySet    [iL_Counter]   := sAdsIkInkStorageTank[iL_Counter].sI_InkDensitySet.fI_Val;
    sR_RemVar_I.sI_CorrectionValue  [iL_Counter]   := sAdsIkInkStorageTank[iL_Counter].sI_CorrectionValue.fI_Val;
    sR_RemVar_I.sI_WarningLevelSet  [iL_Counter]   := sAdsIkInkStorageTank[iL_Counter].sI_WarningLevelSet.fI_Val;
    sR_RemVar_I.sI_ErrorlevelSet    [iL_Counter]   := sAdsIkInkStorageTank[iL_Counter].sI_ErrorlevelSet.fI_Val;

    (*Varnish parameter*)
    sR_RemVar_I.lR_VarParamScannerId[iL_Counter]   := sAdsIkInkStorageTank[iL_Counter].sI_InkParameter.iScannerId;
    sR_RemVar_I.iR_VarParamIndex    [iL_Counter]   := sAdsIkInkStorageTank[iL_Counter].sI_InkParameter.iIndex;
    sR_RemVar_I.fR_VarParamTemp     [iL_Counter]   := sAdsIkInkStorageTank[iL_Counter].sI_InkParameter.sTemperature.fI_Val;
    sR_RemVar_I.fR_VarParamMenc     [iL_Counter]   := sAdsIkInkStorageTank[iL_Counter].sI_InkParameter.sMeniscus.fI_Val;
    sR_RemVar_I.aR_VarParamWaveform [iL_Counter]   := sAdsIkInkStorageTank[iL_Counter].sI_InkParameter.aWaveform;
    sR_RemVar_I.iR_VarParamTimer    [iL_Counter]   := sAdsIkInkStorageTank[iL_Counter].sI_InkParameter.iTimer;
    sR_RemVar_I.fR_VarParamDensity  [iL_Counter]   := sAdsIkInkStorageTank[iL_Counter].sI_InkParameter.sDensity.fI_Val;
    sR_RemVar_I.fR_VarParamViscosity[iL_Counter]   := sAdsIkInkStorageTank[iL_Counter].sI_InkParameter.sViscosity.fI_Val;
    sR_RemVar_I.iR_VarParamColorId  [iL_Counter]   := sAdsIkInkStorageTank[iL_Counter].sI_InkParameter.iColorId;
    FOR iL_Counter2 := 1 TO 10 DO
      sR_RemVar_I.bR_VarParamCompatibility[iL_Counter, iL_Counter2] := sAdsIkInkStorageTank[iL_Counter].sI_InkParameter.bCompatibility[iL_Counter2];
    END_FOR;

    sR_RemVar_I.aI_CalibrateFrameText1[iL_Counter] := sAdsIkInkStorageTank[iL_Counter].aI_CalibrateFrameText1;
    sR_RemVar_I.aI_CalibrateFrameText2[iL_Counter] := sAdsIkInkStorageTank[iL_Counter].aI_CalibrateFrameText2;

    sR_RemVar_I.fR_BalanceOffset[iL_Counter] := fL_BalanceOffset[iL_Counter];
  END_FOR;

END_IF;
END_ACTION

ACTION Simulate:
FOR iL_CounterDgas := 1 TO iCIk_NB_DGAS DO
  fb_DgasMencContr[iL_CounterDgas].iI_ActValue := LREAL_TO_INT(fb_DgasMencContr[iL_CounterDgas].pSetValue * fb_DgasMencContr[iL_CounterDgas].fR_ConvAdsToLocal);

  sAdsIkDgas[iL_CounterDgas].bI_Enable := TRUE;
END_FOR

FOR iL_CounterMenc := 1 TO iCIk_NB_MENC_STA DO
  fb_MeniscusMencContr[iL_CounterMenc].iI_ActValue := LREAL_TO_INT(fb_MeniscusMencContr[iL_CounterMenc].pSetValue * fb_MeniscusMencContr[iL_CounterMenc].fR_ConvAdsToLocal);

  sAdsIkMenc[iL_CounterMenc].bI_Enable := TRUE;
END_FOR

bIKn_TankCleanerLevelEmpty := TRUE;
bIKn_TankRefuseLevelFull   := TRUE;

FOR iL_Counter := 1 TO iCIk_NB_TEMP_HYS DO
  fb_TempControllerHys[iL_Counter].iI_ActValue := DINT_TO_INT(fb_TempControllerHys[iL_Counter].pSetValue);
END_FOR
END_ACTION

ACTION Visu:
(*call visu controls*)
fb_VisuDgasMencController    (sI_Ary_Fb := fb_DgasMencContr    , sI_Ary_Ads := sAdsIkDgas);
fb_VisuMeniscusMencController(sI_Ary_Fb := fb_MeniscusMencContr, sI_Ary_Ads := sAdsIkMenc);
END_ACTION

END_PROGRAM

(* stored: Version 1.1.0.1, ProductVersion 3.1.4024.11
   POU PRG_INK: Id {afcab994-f568-4c43-8a58-3d4d653d253f}, SpecialFunc None
   Action AutoFlushingDevice: Id {6627fb9e-33a2-468a-baa9-49ad7fdee6fb}
   Action Init: Id {3df6df47-00b1-4dfe-b031-bbb8c830433a}
   Action Mapping: Id {b4c298ef-206d-4e7f-8ff8-e09dc27d129d}
   Action RemVar: Id {411712ed-e22a-4c35-81dc-55a2048f7425}
   Action Simulate: Id {508ed5c3-b0e3-425a-a7cb-2e0393f6db76}
   Action Visu: Id {6ca6bb5d-a511-4764-b7c7-2f50776ed47f} *)
